LIN {X 0,Y 498.78,Z 857.029,A -85,B 0,C 180,E1 14801.152,E2 14801.152} C_VEL
LIN {X 0,Y 480.822,Z 920.353,A -85,B 0,C 180,E1 14806.511,E2 14806.511} C_VEL
LIN {X 0,Y 463.831,Z 974.464,A -85,B 0,C 180,E1 14813.724,E2 14813.724} C_VEL
LIN {X 0,Y 451.235,Z 1016.767,A -85,B 0,C 180,E1 14822.478,E2 14822.478} C_VEL
LIN {X 0,Y 444.81,Z 1044.673,A -85,B 0,C 180,E1 14831.852,E2 14831.852} C_VEL
LIN {X 0,Y 443.283,Z 1056.769,A -85,B 0,C 180,E1 14839.155,E2 14839.155} C_VEL
LIN {X 0,Y 443.188,Z 1061.056,A -85,B 0,C 180,E1 14847.74,E2 14847.74} C_VEL
LIN {X 0,Y 443.49,Z 1055.308,A -85,B 0,C 180,E1 14855.887,E2 14855.887} C_VEL
LIN {X 0,Y 445.923,Z 1037.781,A -85,B 0,C 180,E1 14864.776,E2 14864.776} C_VEL
LIN {X 0,Y 454.067,Z 1004.775,A -85,B 0,C 180,E1 14874.148,E2 14874.148} C_VEL
LIN {X 0,Y 467.703,Z 958.825,A -85,B 0,C 180,E1 14882.342,E2 14882.342} C_VEL
LIN {X 0,Y 484.897,Z 900.577,A -85,B 0,C 180,E1 14889.005,E2 14889.005} C_VEL
LIN {X 0,Y 501.352,Z 834.705,A -85,B 0,C 180,E1 14893.779,E2 14893.779} C_VEL
LIN {X 0,Y 509.754,Z 781.732,A -85,B 0,C 180,E1 14896.414,E2 14896.414} C_VEL
LIN {X 0,Y 485.015,Z 728.25,A -85,B 0,C 180,E1 14902.556,E2 14902.556} C_VEL
LIN {X 0,Y 455.384,Z 683.445,A -85,B 0,C 180,E1 14909.799,E2 14909.799} C_VEL
LIN {X 0,Y 441.694,Z 663.19,A -85,B 0,C 180,E1 14914.159,E2 14914.159} C_VEL
LIN {X 0,Y 442.478,Z 663.19,A -85,B 0,C 180,E1 14925.114,E2 14925.114} C_VEL
LIN {X 0,Y 442.609,Z 663.19,A -85,B 0,C 180,E1 14929.547,E2 14929.547} C_VEL
LIN {X 0,Y 434.436,Z 663.19,A -85,B 0,C 180,E1 14934.054,E2 14934.054} C_VEL
LIN {X 0,Y 434.643,Z 663.19,A -85,B 0,C 180,E1 14943.024,E2 14943.024} C_VEL
LIN {X 0,Y 434.152,Z 663.19,A -85,B 0,C 180,E1 14953.157,E2 14953.157} C_VEL
LIN {X 0,Y 433.829,Z 664.9,A -85,B 0,C 180,E1 14960.435,E2 14960.435} C_VEL
LIN {X 0,Y 463.212,Z 704.391,A -85,B 0,C 180,E1 14969.385,E2 14969.385} C_VEL
LIN {X 0,Y 491.827,Z 754.152,A -85,B 0,C 180,E1 14976.332,E2 14976.332} C_VEL
LIN {X 0,Y 505.339,Z 789.902,A -85,B 0,C 180,E1 14980.076,E2 14980.076} C_VEL
LIN {X 0,Y 490.914,Z 859.853,A -85,B 0,C 180,E1 14983.564,E2 14983.564} C_VEL
LIN {X 0,Y 473.096,Z 925.13,A -85,B 0,C 180,E1 14988.962,E2 14988.962} C_VEL
LIN {X 0,Y 456.226,Z 980.153,A -85,B 0,C 180,E1 14996.149,E2 14996.149} C_VEL
LIN {X 0,Y 443.812,Z 1022.566,A -85,B 0,C 180,E1 15004.717,E2 15004.717} C_VEL
LIN {X 0,Y 436.833,Z 1052.193,A -85,B 0,C 180,E1 15014.394,E2 15014.394} C_VEL
LIN {X 0,Y 435.277,Z 1066.186,A -85,B 0,C 180,E1 15022.997,E2 15022.997} C_VEL
LIN {X 0,Y 435.491,Z 1069.578,A -85,B 0,C 180,E1 15030.998,E2 15030.998} C_VEL
LIN {X 0,Y 435.549,Z 1062.657,A -85,B 0,C 180,E1 15040.026,E2 15040.026} C_VEL
LIN {X 0,Y 439.139,Z 1042.2,A -85,B 0,C 180,E1 15049.675,E2 15049.675} C_VEL
LIN {X 0,Y 448.991,Z 1006.051,A -85,B 0,C 180,E1 15059.323,E2 15059.323} C_VEL
LIN {X 0,Y 464.337,Z 958.152,A -85,B 0,C 180,E1 15067.421,E2 15067.421} C_VEL
LIN {X 0,Y 482.711,Z 899.542,A -85,B 0,C 180,E1 15073.825,E2 15073.825} C_VEL
LIN {X 0,Y 500.489,Z 832.188,A -85,B 0,C 180,E1 15078.418,E2 15078.418} C_VEL
LIN {X 0,Y 508.3,Z 786.213,A -85,B 0,C 180,E1 15080.591,E2 15080.591} C_VEL
LIN {X 0,Y 484.766,Z 736.368,A -85,B 0,C 180,E1 15087.094,E2 15087.094} C_VEL
LIN {X 0,Y 459.06,Z 697.737,A -85,B 0,C 180,E1 15094.521,E2 15094.521} C_VEL
LIN {X 0,Y 442.234,Z 676.205,A -85,B 0,C 180,E1 15101.078,E2 15101.078} C_VEL
LIN {X 0,Y 436.452,Z 669.072,A -85,B 0,C 180,E1 15104.118,E2 15104.118} C_VEL
LIN {X 0,Y 434.075,Z 663.19,A -85,B 0,C 180,E1 15106.326,E2 15106.326} C_VEL
LIN {X 0,Y 434.65,Z 663.19,A -85,B 0,C 180,E1 15116.976,E2 15116.976} C_VEL
LIN {X 0,Y 434.433,Z 663.19,A -85,B 0,C 180,E1 15125.837,E2 15125.837} C_VEL
LIN {X 0,Y 434.503,Z 665.136,A -85,B 0,C 180,E1 15131.669,E2 15131.669} C_VEL
LIN {X 0,Y 447.525,Z 682.237,A -85,B 0,C 180,E1 15138.325,E2 15138.325} C_VEL
LIN {X 0,Y 470.261,Z 712.636,A -85,B 0,C 180,E1 15146.001,E2 15146.001} C_VEL
LIN {X 0,Y 495.719,Z 757.278,A -85,B 0,C 180,E1 15153.091,E2 15153.091} C_VEL
LIN {X 0,Y 507.94,Z 791.531,A -85,B 0,C 180,E1 15157.02,E2 15157.02} C_VEL
LIN {X 0,Y 492.588,Z 859.65,A -85,B 0,C 180,E1 15160.625,E2 15160.625} C_VEL
LIN {X 0,Y 474.034,Z 922.35,A -85,B 0,C 180,E1 15166.06,E2 15166.06} C_VEL
LIN {X 0,Y 456.421,Z 976.246,A -85,B 0,C 180,E1 15173.424,E2 15173.424} C_VEL
LIN {X 0,Y 443.207,Z 1018.661,A -85,B 0,C 180,E1 15182.49,E2 15182.49} C_VEL
LIN {X 0,Y 436.635,Z 1046.422,A -85,B 0,C 180,E1 15192.309,E2 15192.309} C_VEL
LIN {X 0,Y 435.14,Z 1058.726,A -85,B 0,C 180,E1 15200.977,E2 15200.977} C_VEL
LIN {X 0,Y 435.281,Z 1060.917,A -85,B 0,C 180,E1 15209.001,E2 15209.001} C_VEL
LIN {X 0,Y 435.779,Z 1052.584,A -85,B 0,C 180,E1 15218.001,E2 15218.001} C_VEL
LIN {X 0,Y 440.317,Z 1029.675,A -85,B 0,C 180,E1 15227.941,E2 15227.941} C_VEL
LIN {X 0,Y 450.604,Z 992.208,A -85,B 0,C 180,E1 15237.291,E2 15237.291} C_VEL
LIN {X 0,Y 466.318,Z 941.94,A -85,B 0,C 180,E1 15245.186,E2 15245.186} C_VEL
LIN {X 0,Y 484.277,Z 880.392,A -85,B 0,C 180,E1 15251.389,E2 15251.389} C_VEL
LIN {X 0,Y 500.471,Z 812.301,A -85,B 0,C 180,E1 15255.622,E2 15255.622} C_VEL
LIN {X 0,Y 503.68,Z 784.382,A -85,B 0,C 180,E1 15257.043,E2 15257.043} C_VEL
LIN {X 0,Y 480.044,Z 732.332,A -85,B 0,C 180,E1 15263.229,E2 15263.229} C_VEL
LIN {X 0,Y 451.395,Z 688.691,A -85,B 0,C 180,E1 15270.571,E2 15270.571} C_VEL
LIN {X 0,Y 433.747,Z 663.19,A -85,B 0,C 180,E1 15276.72,E2 15276.72} C_VEL
LIN {X 0,Y 434.648,Z 663.19,A -85,B 0,C 180,E1 15286.903,E2 15286.903} C_VEL
LIN {X 0,Y 434.436,Z 663.19,A -85,B 0,C 180,E1 15294.054,E2 15294.054} C_VEL
LIN {X 0,Y 426.744,Z 663.19,A -85,B 0,C 180,E1 15298.697,E2 15298.697} C_VEL
LIN {X 0,Y 426.485,Z 663.19,A -85,B 0,C 180,E1 15307.178,E2 15307.178} C_VEL
LIN {X 0,Y 425.974,Z 665.123,A -85,B 0,C 180,E1 15317.653,E2 15317.653} C_VEL
LIN {X 0,Y 448.471,Z 695.077,A -85,B 0,C 180,E1 15325.749,E2 15325.749} C_VEL
LIN {X 0,Y 474.865,Z 735.267,A -85,B 0,C 180,E1 15332.732,E2 15332.732} C_VEL
LIN {X 0,Y 498.15,Z 786.178,A -85,B 0,C 180,E1 15338.91,E2 15338.91} C_VEL
LIN {X 0,Y 498.656,Z 798.243,A -85,B 0,C 180,E1 15339.698,E2 15339.698} C_VEL
LIN {X 0,Y 483.298,Z 867.659,A -85,B 0,C 180,E1 15343.412,E2 15343.412} C_VEL
LIN {X 0,Y 465.118,Z 930.433,A -85,B 0,C 180,E1 15348.904,E2 15348.904} C_VEL
LIN {X 0,Y 447.9,Z 984.105,A -85,B 0,C 180,E1 15356.257,E2 15356.257} C_VEL
LIN {X 0,Y 435.152,Z 1026.238,A -85,B 0,C 180,E1 15365.249,E2 15365.249} C_VEL
LIN {X 0,Y 428.705,Z 1053.233,A -85,B 0,C 180,E1 15374.616,E2 15374.616} C_VEL
LIN {X 0,Y 427.272,Z 1066.093,A -85,B 0,C 180,E1 15382.865,E2 15382.865} C_VEL
LIN {X 0,Y 427.503,Z 1069.503,A -85,B 0,C 180,E1 15391.017,E2 15391.017} C_VEL
LIN {X 0,Y 427.571,Z 1062.604,A -85,B 0,C 180,E1 15400.215,E2 15400.215} C_VEL
LIN {X 0,Y 431.395,Z 1042.278,A -85,B 0,C 180,E1 15410.009,E2 15410.009} C_VEL
LIN {X 0,Y 441.734,Z 1006.072,A -85,B 0,C 180,E1 15419.853,E2 15419.853} C_VEL
LIN {X 0,Y 458.167,Z 957.186,A -85,B 0,C 180,E1 15428.193,E2 15428.193} C_VEL
LIN {X 0,Y 477.4,Z 897.844,A -85,B 0,C 180,E1 15434.675,E2 15434.675} C_VEL
LIN {X 0,Y 495.435,Z 831.195,A -85,B 0,C 180,E1 15439.185,E2 15439.185} C_VEL
LIN {X 0,Y 502.744,Z 789.669,A -85,B 0,C 180,E1 15441.181,E2 15441.181} C_VEL
LIN {X 0,Y 479.872,Z 740.348,A -85,B 0,C 180,E1 15447.876,E2 15447.876} C_VEL
LIN {X 0,Y 455.268,Z 702.676,A -85,B 0,C 180,E1 15455.415,E2 15455.415} C_VEL
LIN {X 0,Y 436.885,Z 678.131,A -85,B 0,C 180,E1 15463.336,E2 15463.336} C_VEL
LIN {X 0,Y 429.602,Z 669.753,A -85,B 0,C 180,E1 15468.168,E2 15468.168} C_VEL
LIN {X 0,Y 426.492,Z 663.19,A -85,B 0,C 180,E1 15472.823,E2 15472.823} C_VEL
LIN {X 0,Y 426.967,Z 663.19,A -85,B 0,C 180,E1 15483.034,E2 15483.034} C_VEL
LIN {X 0,Y 426.767,Z 665.544,A -85,B 0,C 180,E1 15486.09,E2 15486.09} C_VEL
LIN {X 0,Y 433.558,Z 674.22,A -85,B 0,C 180,E1 15491.782,E2 15491.782} C_VEL
LIN {X 0,Y 445.568,Z 689.42,A -85,B 0,C 180,E1 15497.959,E2 15497.959} C_VEL
LIN {X 0,Y 468.291,Z 720.914,A -85,B 0,C 180,E1 15505.861,E2 15505.861} C_VEL
LIN {X 0,Y 492.084,Z 764.56,A -85,B 0,C 180,E1 15512.908,E2 15512.908} C_VEL
LIN {X 0,Y 502.331,Z 794.471,A -85,B 0,C 180,E1 15516.421,E2 15516.421} C_VEL
LIN {X 0,Y 486.135,Z 863.156,A -85,B 0,C 180,E1 15520.16,E2 15520.16} C_VEL
LIN {X 0,Y 466.596,Z 926.451,A -85,B 0,C 180,E1 15525.836,E2 15525.836} C_VEL
LIN {X 0,Y 448.604,Z 979.206,A -85,B 0,C 180,E1 15533.316,E2 15533.316} C_VEL
LIN {X 0,Y 435.185,Z 1020.487,A -85,B 0,C 180,E1 15542.49,E2 15542.49} C_VEL
LIN {X 0,Y 428.578,Z 1047.393,A -85,B 0,C 180,E1 15552.497,E2 15552.497} C_VEL
LIN {X 0,Y 427.138,Z 1058.771,A -85,B 0,C 180,E1 15560.807,E2 15560.807} C_VEL
LIN {X 0,Y 427.294,Z 1061.002,A -85,B 0,C 180,E1 15568.983,E2 15568.983} C_VEL
LIN {X 0,Y 427.826,Z 1052.724,A -85,B 0,C 180,E1 15578.15,E2 15578.15} C_VEL
LIN {X 0,Y 432.49,Z 1030.138,A -85,B 0,C 180,E1 15588.183,E2 15588.183} C_VEL
LIN {X 0,Y 442.958,Z 993.681,A -85,B 0,C 180,E1 15597.526,E2 15597.526} C_VEL
LIN {X 0,Y 458.683,Z 945.619,A -85,B 0,C 180,E1 15605.348,E2 15605.348} C_VEL
LIN {X 0,Y 476.882,Z 885.865,A -85,B 0,C 180,E1 15611.617,E2 15611.617} C_VEL
LIN {X 0,Y 494.078,Z 817.022,A -85,B 0,C 180,E1 15616.078,E2 15616.078} C_VEL
LIN {X 0,Y 497.877,Z 787.864,A -85,B 0,C 180,E1 15617.608,E2 15617.608} C_VEL
LIN {X 0,Y 475.449,Z 737.244,A -85,B 0,C 180,E1 15623.826,E2 15623.826} C_VEL
LIN {X 0,Y 446.571,Z 691.869,A -85,B 0,C 180,E1 15631.661,E2 15631.661} C_VEL
LIN {X 0,Y 428.138,Z 668.883,A -85,B 0,C 180,E1 15638.17,E2 15638.17} C_VEL
LIN {X 0,Y 425.795,Z 663.19,A -85,B 0,C 180,E1 15639.686,E2 15639.686} C_VEL
LIN {X 0,Y 426.677,Z 663.19,A -85,B 0,C 180,E1 15648.74,E2 15648.74} C_VEL
LIN {X 0,Y 426.744,Z 663.19,A -85,B 0,C 180,E1 15658.697,E2 15658.697} C_VEL
LIN {X 0,Y 418.627,Z 663.19,A -85,B 0,C 180,E1 15663.379,E2 15663.379} C_VEL
LIN {X 0,Y 418.152,Z 664.953,A -85,B 0,C 180,E1 15674.273,E2 15674.273} C_VEL
LIN {X 0,Y 436.427,Z 689.311,A -85,B 0,C 180,E1 15682.264,E2 15682.264} C_VEL
LIN {X 0,Y 462.637,Z 726.523,A -85,B 0,C 180,E1 15690.038,E2 15690.038} C_VEL
LIN {X 0,Y 487.402,Z 776.2,A -85,B 0,C 180,E1 15696.802,E2 15696.802} C_VEL
LIN {X 0,Y 493.513,Z 797.499,A -85,B 0,C 180,E1 15698.963,E2 15698.963} C_VEL
LIN {X 0,Y 477.824,Z 866.764,A -85,B 0,C 180,E1 15702.657,E2 15702.657} C_VEL
LIN {X 0,Y 458.773,Z 930.381,A -85,B 0,C 180,E1 15708.243,E2 15708.243} C_VEL
LIN {X 0,Y 440.535,Z 985.235,A -85,B 0,C 180,E1 15715.885,E2 15715.885} C_VEL
LIN {X 0,Y 427.488,Z 1026.605,A -85,B 0,C 180,E1 15724.925,E2 15724.925} C_VEL
LIN {X 0,Y 420.634,Z 1054.271,A -85,B 0,C 180,E1 15734.849,E2 15734.849} C_VEL
LIN {X 0,Y 419.279,Z 1066,A -85,B 0,C 180,E1 15742.728,E2 15742.728} C_VEL
LIN {X 0,Y 419.491,Z 1069.428,A -85,B 0,C 180,E1 15751.036,E2 15751.036} C_VEL
LIN {X 0,Y 419.619,Z 1062.554,A -85,B 0,C 180,E1 15760.41,E2 15760.41} C_VEL
LIN {X 0,Y 423.642,Z 1042.363,A -85,B 0,C 180,E1 15770.355,E2 15770.355} C_VEL
LIN {X 0,Y 434.139,Z 1007.297,A -85,B 0,C 180,E1 15780.14,E2 15780.14} C_VEL
LIN {X 0,Y 451.184,Z 958.707,A -85,B 0,C 180,E1 15788.64,E2 15788.64} C_VEL
LIN {X 0,Y 471.074,Z 899.714,A -85,B 0,C 180,E1 15795.218,E2 15795.218} C_VEL
LIN {X 0,Y 490.205,Z 831.579,A -85,B 0,C 180,E1 15799.893,E2 15799.893} C_VEL
LIN {X 0,Y 497.337,Z 793.409,A -85,B 0,C 180,E1 15801.752,E2 15801.752} C_VEL
LIN {X 0,Y 474.61,Z 743.426,A -85,B 0,C 180,E1 15808.811,E2 15808.811} C_VEL
LIN {X 0,Y 450.499,Z 706.201,A -85,B 0,C 180,E1 15816.723,E2 15816.723} C_VEL
LIN {X 0,Y 434.137,Z 684.921,A -85,B 0,C 180,E1 15824.274,E2 15824.274} C_VEL
LIN {X 0,Y 428.274,Z 677.491,A -85,B 0,C 180,E1 15828.434,E2 15828.434} C_VEL
LIN {X 0,Y 423.877,Z 670.721,A -85,B 0,C 180,E1 15833.811,E2 15833.811} C_VEL
LIN {X 0,Y 425.501,Z 672.996,A -85,B 0,C 180,E1 15845.736,E2 15845.736} C_VEL
LIN {X 0,Y 432.732,Z 682.917,A -85,B 0,C 180,E1 15851.934,E2 15851.934} C_VEL
LIN {X 0,Y 447.738,Z 701.689,A -85,B 0,C 180,E1 15859.278,E2 15859.278} C_VEL
LIN {X 0,Y 471.802,Z 738.399,A -85,B 0,C 180,E1 15867.522,E2 15867.522} C_VEL
LIN {X 0,Y 493.23,Z 784.173,A -85,B 0,C 180,E1 15874.336,E2 15874.336} C_VEL
LIN {X 0,Y 496.572,Z 798.512,A -85,B 0,C 180,E1 15875.861,E2 15875.861} C_VEL
LIN {X 0,Y 479.996,Z 865.734,A -85,B 0,C 180,E1 15879.618,E2 15879.618} C_VEL
LIN {X 0,Y 459.786,Z 928.731,A -85,B 0,C 180,E1 15885.396,E2 15885.396} C_VEL
LIN {X 0,Y 441.159,Z 981.112,A -85,B 0,C 180,E1 15893.02,E2 15893.02} C_VEL
LIN {X 0,Y 427.338,Z 1021.674,A -85,B 0,C 180,E1 15902.347,E2 15902.347} C_VEL
LIN {X 0,Y 420.72,Z 1047.399,A -85,B 0,C 180,E1 15912.159,E2 15912.159} C_VEL
LIN {X 0,Y 419.138,Z 1058.816,A -85,B 0,C 180,E1 15920.63,E2 15920.63} C_VEL
LIN {X 0,Y 419.29,Z 1061.086,A -85,B 0,C 180,E1 15928.963,E2 15928.963} C_VEL
LIN {X 0,Y 419.893,Z 1052.861,A -85,B 0,C 180,E1 15938.305,E2 15938.305} C_VEL
LIN {X 0,Y 424.578,Z 1031.01,A -85,B 0,C 180,E1 15948.292,E2 15948.292} C_VEL
LIN {X 0,Y 435.694,Z 993.933,A -85,B 0,C 180,E1 15958.025,E2 15958.025} C_VEL
LIN {X 0,Y 452.484,Z 944.571,A -85,B 0,C 180,E1 15966.125,E2 15966.125} C_VEL
LIN {X 0,Y 471.328,Z 884.634,A -85,B 0,C 180,E1 15972.411,E2 15972.411} C_VEL
LIN {X 0,Y 488.788,Z 816.604,A -85,B 0,C 180,E1 15976.807,E2 15976.807} C_VEL
LIN {X 0,Y 492.112,Z 791.275,A -85,B 0,C 180,E1 15978.192,E2 15978.192} C_VEL
LIN {X 0,Y 470.456,Z 741.37,A -85,B 0,C 180,E1 15984.524,E2 15984.524} C_VEL
LIN {X 0,Y 443.694,Z 698.608,A -85,B 0,C 180,E1 15992.168,E2 15992.168} C_VEL
LIN {X 0,Y 422.122,Z 670.229,A -85,B 0,C 180,E1 16000.454,E2 16000.454} C_VEL
LIN {X 0,Y 418.095,Z 663.19,A -85,B 0,C 180,E1 16003.048,E2 16003.048} C_VEL
LIN {X 0,Y 418.386,Z 663.19,A -85,B 0,C 180,E1 16012.728,E2 16012.728} C_VEL
LIN {X 0,Y 418.464,Z 663.19,A -85,B 0,C 180,E1 16021.062,E2 16021.062} C_VEL
LIN {X 0,Y 418.627,Z 663.19,A -85,B 0,C 180,E1 16023.379,E2 16023.379} C_VEL
LIN {X 0,Y 410.326,Z 663.19,A -85,B 0,C 180,E1 16028.157,E2 16028.157} C_VEL
LIN {X 0,Y 410.695,Z 666.004,A -85,B 0,C 180,E1 16030.134,E2 16030.134} C_VEL
LIN {X 0,Y 417.572,Z 674.992,A -85,B 0,C 180,E1 16034.609,E2 16034.609} C_VEL
LIN {X 0,Y 433.792,Z 695.796,A -85,B 0,C 180,E1 16041.729,E2 16041.729} C_VEL
LIN {X 0,Y 459.528,Z 733.457,A -85,B 0,C 180,E1 16049.722,E2 16049.722} C_VEL
LIN {X 0,Y 482.731,Z 781.872,A -85,B 0,C 180,E1 16056.428,E2 16056.428} C_VEL
LIN {X 0,Y 487.905,Z 799.598,A -85,B 0,C 180,E1 16058.33,E2 16058.33} C_VEL
LIN {X 0,Y 471.492,Z 869.149,A -85,B 0,C 180,E1 16062.121,E2 16062.121} C_VEL
LIN {X 0,Y 451.706,Z 932.866,A -85,B 0,C 180,E1 16067.86,E2 16067.86} C_VEL
LIN {X 0,Y 432.989,Z 986.936,A -85,B 0,C 180,E1 16075.601,E2 16075.601} C_VEL
LIN {X 0,Y 419.444,Z 1028.165,A -85,B 0,C 180,E1 16084.923,E2 16084.923} C_VEL
LIN {X 0,Y 412.534,Z 1055.151,A -85,B 0,C 180,E1 16095.09,E2 16095.09} C_VEL
LIN {X 0,Y 411.199,Z 1067.647,A -85,B 0,C 180,E1 16104.711,E2 16104.711} C_VEL
LIN {X 0,Y 411.152,Z 1068.842,A -85,B 0,C 180,E1 16113.172,E2 16113.172} C_VEL
LIN {X 0,Y 412.384,Z 1058.853,A -85,B 0,C 180,E1 16123.08,E2 16123.08} C_VEL
LIN {X 0,Y 417.766,Z 1034.302,A -85,B 0,C 180,E1 16133.534,E2 16133.534} C_VEL
LIN {X 0,Y 430.738,Z 996.165,A -85,B 0,C 180,E1 16143.071,E2 16143.071} C_VEL
LIN {X 0,Y 450.189,Z 943.725,A -85,B 0,C 180,E1 16151.313,E2 16151.313} C_VEL
LIN {X 0,Y 470.83,Z 882.841,A -85,B 0,C 180,E1 16157.342,E2 16157.342} C_VEL
LIN {X 0,Y 489.351,Z 812.57,A -85,B 0,C 180,E1 16161.584,E2 16161.584} C_VEL
LIN {X 0,Y 491.697,Z 796.347,A -85,B 0,C 180,E1 16162.434,E2 16162.434} C_VEL
LIN {X 0,Y 469.974,Z 748.012,A -85,B 0,C 180,E1 16169.534,E2 16169.534} C_VEL
LIN {X 0,Y 447.711,Z 712.682,A -85,B 0,C 180,E1 16177.295,E2 16177.295} C_VEL
LIN {X 0,Y 431.971,Z 691.832,A -85,B 0,C 180,E1 16184.959,E2 16184.959} C_VEL
LIN {X 0,Y 426.531,Z 684.771,A -85,B 0,C 180,E1 16189.081,E2 16189.081} C_VEL
LIN {X 0,Y 422.626,Z 678.518,A -85,B 0,C 180,E1 16194.31,E2 16194.31} C_VEL
LIN {X 0,Y 424.354,Z 680.93,A -85,B 0,C 180,E1 16205.558,E2 16205.558} C_VEL
LIN {X 0,Y 432.326,Z 691.884,A -85,B 0,C 180,E1 16212.331,E2 16212.331} C_VEL
LIN {X 0,Y 447.389,Z 711.911,A -85,B 0,C 180,E1 16219.68,E2 16219.68} C_VEL
LIN {X 0,Y 469.419,Z 746.964,A -85,B 0,C 180,E1 16227.508,E2 16227.508} C_VEL
LIN {X 0,Y 489.261,Z 791.653,A -85,B 0,C 180,E1 16234.198,E2 16234.198} C_VEL
LIN {X 0,Y 490.644,Z 803.508,A -85,B 0,C 180,E1 16235.326,E2 16235.326} C_VEL
LIN {X 0,Y 473.328,Z 870.264,A -85,B 0,C 180,E1 16239.203,E2 16239.203} C_VEL
LIN {X 0,Y 452.36,Z 932.822,A -85,B 0,C 180,E1 16245.151,E2 16245.151} C_VEL
LIN {X 0,Y 433.01,Z 984.809,A -85,B 0,C 180,E1 16253.078,E2 16253.078} C_VEL
LIN {X 0,Y 419.173,Z 1023.727,A -85,B 0,C 180,E1 16262.465,E2 16262.465} C_VEL
LIN {X 0,Y 412.585,Z 1048.87,A -85,B 0,C 180,E1 16272.634,E2 16272.634} C_VEL
LIN {X 0,Y 411.141,Z 1058.862,A -85,B 0,C 180,E1 16280.446,E2 16280.446} C_VEL
LIN {X 0,Y 411.285,Z 1061.171,A -85,B 0,C 180,E1 16288.943,E2 16288.943} C_VEL
LIN {X 0,Y 411.961,Z 1052.997,A -85,B 0,C 180,E1 16298.466,E2 16298.466} C_VEL
LIN {X 0,Y 416.812,Z 1031.202,A -85,B 0,C 180,E1 16308.645,E2 16308.645} C_VEL
LIN {X 0,Y 428.484,Z 994.183,A -85,B 0,C 180,E1 16318.539,E2 16318.539} C_VEL
LIN {X 0,Y 445.848,Z 945.171,A -85,B 0,C 180,E1 16326.709,E2 16326.709} C_VEL
LIN {X 0,Y 465.527,Z 884.677,A -85,B 0,C 180,E1 16333.114,E2 16333.114} C_VEL
LIN {X 0,Y 483.714,Z 815.532,A -85,B 0,C 180,E1 16337.586,E2 16337.586} C_VEL
LIN {X 0,Y 486.452,Z 795.07,A -85,B 0,C 180,E1 16338.728,E2 16338.728} C_VEL
LIN {X 0,Y 465.506,Z 745.361,A -85,B 0,C 180,E1 16345.233,E2 16345.233} C_VEL
LIN {X 0,Y 440.008,Z 704.189,A -85,B 0,C 180,E1 16352.948,E2 16352.948} C_VEL
LIN {X 0,Y 420.1,Z 677.619,A -85,B 0,C 180,E1 16360.911,E2 16360.911} C_VEL
LIN {X 0,Y 413.018,Z 669.205,A -85,B 0,C 180,E1 16364.981,E2 16364.981} C_VEL
LIN {X 0,Y 410.543,Z 663.19,A -85,B 0,C 180,E1 16367.316,E2 16367.316} C_VEL
LIN {X 0,Y 410.76,Z 663.19,A -85,B 0,C 180,E1 16378.964,E2 16378.964} C_VEL
LIN {X 0,Y 410.326,Z 663.19,A -85,B 0,C 180,E1 16388.157,E2 16388.157} C_VEL
LIN {X 0,Y 410.731,Z 676.091,A -85,B 0,C 180,E1 16390.981,E2 16390.981} C_VEL
LIN {X 0,Y 420.44,Z 687.719,A -85,B 0,C 180,E1 16396.607,E2 16396.607} C_VEL
LIN {X 0,Y 443.836,Z 719.972,A -85,B 0,C 180,E1 16405.533,E2 16405.533} C_VEL
LIN {X 0,Y 467.876,Z 762.883,A -85,B 0,C 180,E1 16412.837,E2 16412.837} C_VEL
LIN {X 0,Y 482.174,Z 802.573,A -85,B 0,C 180,E1 16417.725,E2 16417.725} C_VEL
LIN {X 0,Y 465.103,Z 871.898,A -85,B 0,C 180,E1 16421.598,E2 16421.598} C_VEL
LIN {X 0,Y 444.653,Z 935.254,A -85,B 0,C 180,E1 16427.449,E2 16427.449} C_VEL
LIN {X 0,Y 425.464,Z 988.588,A -85,B 0,C 180,E1 16435.297,E2 16435.297} C_VEL
LIN {X 0,Y 411.411,Z 1029.584,A -85,B 0,C 180,E1 16444.921,E2 16444.921} C_VEL
LIN {X 0,Y 404.653,Z 1055.033,A -85,B 0,C 180,E1 16454.793,E2 16454.793} C_VEL
LIN {X 0,Y 403.207,Z 1067.552,A -85,B 0,C 180,E1 16464.605,E2 16464.605} C_VEL
LIN {X 0,Y 403.122,Z 1068.654,A -85,B 0,C 180,E1 16473.483,E2 16473.483} C_VEL
LIN {X 0,Y 404.467,Z 1058.614,A -85,B 0,C 180,E1 16483.455,E2 16483.455} C_VEL
LIN {X 0,Y 410.185,Z 1034.297,A -85,B 0,C 180,E1 16493.996,E2 16493.996} C_VEL
LIN {X 0,Y 423.8,Z 996.205,A -85,B 0,C 180,E1 16503.684,E2 16503.684} C_VEL
LIN {X 0,Y 443.931,Z 944.043,A -85,B 0,C 180,E1 16511.989,E2 16511.989} C_VEL
LIN {X 0,Y 465.564,Z 882.508,A -85,B 0,C 180,E1 16518.116,E2 16518.116} C_VEL
LIN {X 0,Y 484.304,Z 813.467,A -85,B 0,C 180,E1 16522.305,E2 16522.305} C_VEL
LIN {X 0,Y 486.328,Z 800.34,A -85,B 0,C 180,E1 16522.999,E2 16522.999} C_VEL
LIN {X 0,Y 465.605,Z 752.891,A -85,B 0,C 180,E1 16530.207,E2 16530.207} C_VEL
LIN {X 0,Y 444.55,Z 718.47,A -85,B 0,C 180,E1 16538.05,E2 16538.05} C_VEL
LIN {X 0,Y 427.604,Z 694.207,A -85,B 0,C 180,E1 16547.425,E2 16547.425} C_VEL
LIN {X 0,Y 421.409,Z 686.303,A -85,B 0,C 180,E1 16554.812,E2 16554.812} C_VEL
LIN {X 0,Y 423.218,Z 688.807,A -85,B 0,C 180,E1 16565.379,E2 16565.379} C_VEL
LIN {X 0,Y 433.701,Z 702.296,A -85,B 0,C 180,E1 16573.706,E2 16573.706} C_VEL
LIN {X 0,Y 453.095,Z 731.195,A -85,B 0,C 180,E1 16582.505,E2 16582.505} C_VEL
LIN {X 0,Y 474.432,Z 771.075,A -85,B 0,C 180,E1 16590.101,E2 16590.101} C_VEL
LIN {X 0,Y 485.587,Z 804.638,A -85,B 0,C 180,E1 16594.61,E2 16594.61} C_VEL
LIN {X 0,Y 467.66,Z 871.488,A -85,B 0,C 180,E1 16598.531,E2 16598.531} C_VEL
LIN {X 0,Y 446.2,Z 933.313,A -85,B 0,C 180,E1 16604.475,E2 16604.475} C_VEL
LIN {X 0,Y 426.147,Z 985.009,A -85,B 0,C 180,E1 16612.456,E2 16612.456} C_VEL
LIN {X 0,Y 411.786,Z 1023.681,A -85,B 0,C 180,E1 16621.928,E2 16621.928} C_VEL
LIN {X 0,Y 404.717,Z 1048.925,A -85,B 0,C 180,E1 16632.312,E2 16632.312} C_VEL
LIN {X 0,Y 402.974,Z 1060.342,A -85,B 0,C 180,E1 16642.431,E2 16642.431} C_VEL
LIN {X 0,Y 403.105,Z 1060.411,A -85,B 0,C 180,E1 16651.077,E2 16651.077} C_VEL
LIN {X 0,Y 404.769,Z 1049.772,A -85,B 0,C 180,E1 16660.796,E2 16660.796} C_VEL
LIN {X 0,Y 410.596,Z 1025.231,A -85,B 0,C 180,E1 16671.105,E2 16671.105} C_VEL
LIN {X 0,Y 423.742,Z 987.027,A -85,B 0,C 180,E1 16680.596,E2 16680.596} C_VEL
LIN {X 0,Y 442.82,Z 935.693,A -85,B 0,C 180,E1 16688.611,E2 16688.611} C_VEL
LIN {X 0,Y 462.857,Z 875.092,A -85,B 0,C 180,E1 16694.614,E2 16694.614} C_VEL
LIN {X 0,Y 480.805,Z 804.571,A -85,B 0,C 180,E1 16698.855,E2 16698.855} C_VEL
LIN {X 0,Y 473.443,Z 777.578,A -85,B 0,C 180,E1 16701.918,E2 16701.918} C_VEL
LIN {X 0,Y 449.835,Z 730.158,A -85,B 0,C 180,E1 16709.29,E2 16709.29} C_VEL
LIN {X 0,Y 425.035,Z 693.221,A -85,B 0,C 180,E1 16718.14,E2 16718.14} C_VEL
LIN {X 0,Y 411.665,Z 676.93,A -85,B 0,C 180,E1 16725.204,E2 16725.204} C_VEL
LIN {X 0,Y 407.068,Z 670.401,A -85,B 0,C 180,E1 16729.009,E2 16729.009} C_VEL
LIN {X 0,Y 402.76,Z 663.19,A -85,B 0,C 180,E1 16738.944,E2 16738.944} C_VEL
LIN {X 0,Y 409.313,Z 673.724,A -85,B 0,C 180,E1 16749.85,E2 16749.85} C_VEL
LIN {X 0,Y 410.731,Z 676.091,A -85,B 0,C 180,E1 16750.981,E2 16750.981} C_VEL
LIN {X 0,Y 413.955,Z 689.296,A -85,B 0,C 180,E1 16753.73,E2 16753.73} C_VEL
LIN {X 0,Y 432.831,Z 714.723,A -85,B 0,C 180,E1 16762.27,E2 16762.27} C_VEL
LIN {X 0,Y 456.296,Z 753.371,A -85,B 0,C 180,E1 16770.092,E2 16770.092} C_VEL
LIN {X 0,Y 476.397,Z 803.084,A -85,B 0,C 180,E1 16776.904,E2 16776.904} C_VEL
LIN {X 0,Y 458.764,Z 874.617,A -85,B 0,C 180,E1 16781.058,E2 16781.058} C_VEL
LIN {X 0,Y 437.817,Z 937.111,A -85,B 0,C 180,E1 16786.964,E2 16786.964} C_VEL
LIN {X 0,Y 418.137,Z 989.697,A -85,B 0,C 180,E1 16794.898,E2 16794.898} C_VEL
LIN {X 0,Y 403.944,Z 1029.428,A -85,B 0,C 180,E1 16804.424,E2 16804.424} C_VEL
LIN {X 0,Y 396.793,Z 1054.914,A -85,B 0,C 180,E1 16814.484,E2 16814.484} C_VEL
LIN {X 0,Y 395.198,Z 1067.457,A -85,B 0,C 180,E1 16824.496,E2 16824.496} C_VEL
LIN {X 0,Y 395.164,Z 1068.706,A -85,B 0,C 180,E1 16833.3,E2 16833.3} C_VEL
LIN {X 0,Y 396.434,Z 1059.26,A -85,B 0,C 180,E1 16843.269,E2 16843.269} C_VEL
LIN {X 0,Y 402.114,Z 1035.962,A -85,B 0,C 180,E1 16853.916,E2 16853.916} C_VEL
LIN {X 0,Y 416.406,Z 997.571,A -85,B 0,C 180,E1 16864.05,E2 16864.05} C_VEL
LIN {X 0,Y 436.712,Z 947.032,A -85,B 0,C 180,E1 16872.338,E2 16872.338} C_VEL
LIN {X 0,Y 458.953,Z 886.124,A -85,B 0,C 180,E1 16878.6,E2 16878.6} C_VEL
LIN {X 0,Y 478.498,Z 817.793,A -85,B 0,C 180,E1 16882.876,E2 16882.876} C_VEL
LIN {X 0,Y 480.604,Z 803.229,A -85,B 0,C 180,E1 16883.719,E2 16883.719} C_VEL
LIN {X 0,Y 460.9,Z 756.777,A -85,B 0,C 180,E1 16891.051,E2 16891.051} C_VEL
LIN {X 0,Y 439.898,Z 721.858,A -85,B 0,C 180,E1 16899.53,E2 16899.53} C_VEL
LIN {X 0,Y 425.574,Z 701.589,A -85,B 0,C 180,E1 16908.207,E2 16908.207} C_VEL
LIN {X 0,Y 420.437,Z 694.25,A -85,B 0,C 180,E1 16914.799,E2 16914.799} C_VEL
LIN {X 0,Y 422.132,Z 696.769,A -85,B 0,C 180,E1 16925.264,E2 16925.264} C_VEL
LIN {X 0,Y 432.221,Z 710.344,A -85,B 0,C 180,E1 16933.56,E2 16933.56} C_VEL
LIN {X 0,Y 450.62,Z 738.529,A -85,B 0,C 180,E1 16942.239,E2 16942.239} C_VEL
LIN {X 0,Y 470.322,Z 777.205,A -85,B 0,C 180,E1 16949.724,E2 16949.724} C_VEL
LIN {X 0,Y 480.13,Z 808.043,A -85,B 0,C 180,E1 16953.982,E2 16953.982} C_VEL
LIN {X 0,Y 461.448,Z 874.696,A -85,B 0,C 180,E1 16957.989,E2 16957.989} C_VEL
LIN {X 0,Y 439.224,Z 935.955,A -85,B 0,C 180,E1 16964.059,E2 16964.059} C_VEL
LIN {X 0,Y 418.391,Z 987.576,A -85,B 0,C 180,E1 16972.293,E2 16972.293} C_VEL
LIN {X 0,Y 403.606,Z 1025.751,A -85,B 0,C 180,E1 16982.046,E2 16982.046} C_VEL
LIN {X 0,Y 396.627,Z 1050.144,A -85,B 0,C 180,E1 16992.66,E2 16992.66} C_VEL
LIN {X 0,Y 394.971,Z 1060.402,A -85,B 0,C 180,E1 17002.277,E2 17002.277} C_VEL
LIN {X 0,Y 395.123,Z 1060.507,A -85,B 0,C 180,E1 17011.099,E2 17011.099} C_VEL
LIN {X 0,Y 396.818,Z 1049.92,A -85,B 0,C 180,E1 17021.015,E2 17021.015} C_VEL
LIN {X 0,Y 402.98,Z 1025.433,A -85,B 0,C 180,E1 17031.524,E2 17031.524} C_VEL
LIN {X 0,Y 417.052,Z 986.302,A -85,B 0,C 180,E1 17041.372,E2 17041.372} C_VEL
LIN {X 0,Y 436.639,Z 935.624,A -85,B 0,C 180,E1 17049.33,E2 17049.33} C_VEL
LIN {X 0,Y 457.62,Z 874.08,A -85,B 0,C 180,E1 17055.433,E2 17055.433} C_VEL
LIN {X 0,Y 475.423,Z 803.146,A -85,B 0,C 180,E1 17059.765,E2 17059.765} C_VEL
LIN {X 0,Y 456.44,Z 755.227,A -85,B 0,C 180,E1 17066.464,E2 17066.464} C_VEL
LIN {X 0,Y 433.063,Z 715.031,A -85,B 0,C 180,E1 17074.44,E2 17074.44} C_VEL
LIN {X 0,Y 412.369,Z 686.154,A -85,B 0,C 180,E1 17084.136,E2 17084.136} C_VEL
LIN {X 0,Y 405.271,Z 677.94,A -85,B 0,C 180,E1 17089.777,E2 17089.777} C_VEL
LIN {X 0,Y 401.557,Z 671.088,A -85,B 0,C 180,E1 17098.941,E2 17098.941} C_VEL
LIN {X 0,Y 408.136,Z 681.783,A -85,B 0,C 180,E1 17109.733,E2 17109.733} C_VEL
LIN {X 0,Y 413.955,Z 689.296,A -85,B 0,C 180,E1 17113.73,E2 17113.73} C_VEL
LIN {X 0,Y 417.622,Z 703.934,A -85,B 0,C 180,E1 17116.302,E2 17116.302} C_VEL
LIN {X 0,Y 438.689,Z 734.782,A -85,B 0,C 180,E1 17124.963,E2 17124.963} C_VEL
LIN {X 0,Y 459.758,Z 775.667,A -85,B 0,C 180,E1 17132.164,E2 17132.164} C_VEL
LIN {X 0,Y 470.533,Z 810.03,A -85,B 0,C 180,E1 17136.533,E2 17136.533} C_VEL
LIN {X 0,Y 452.455,Z 877.351,A -85,B 0,C 180,E1 17140.504,E2 17140.504} C_VEL
LIN {X 0,Y 430.526,Z 940.237,A -85,B 0,C 180,E1 17146.621,E2 17146.621} C_VEL
LIN {X 0,Y 410.211,Z 992.147,A -85,B 0,C 180,E1 17154.76,E2 17154.76} C_VEL
LIN {X 0,Y 395.501,Z 1031.923,A -85,B 0,C 180,E1 17164.757,E2 17164.757} C_VEL
LIN {X 0,Y 388.473,Z 1056.745,A -85,B 0,C 180,E1 17175.302,E2 17175.302} C_VEL
LIN {X 0,Y 387.2,Z 1067.362,A -85,B 0,C 180,E1 17184.382,E2 17184.382} C_VEL
LIN {X 0,Y 387.17,Z 1068.638,A -85,B 0,C 180,E1 17193.369,E2 17193.369} C_VEL
LIN {X 0,Y 388.492,Z 1059.213,A -85,B 0,C 180,E1 17203.545,E2 17203.545} C_VEL
LIN {X 0,Y 394.819,Z 1035.088,A -85,B 0,C 180,E1 17214.714,E2 17214.714} C_VEL
LIN {X 0,Y 409.515,Z 997.615,A -85,B 0,C 180,E1 17224.704,E2 17224.704} C_VEL
LIN {X 0,Y 430.727,Z 946.955,A -85,B 0,C 180,E1 17233.1,E2 17233.1} C_VEL
LIN {X 0,Y 453.64,Z 886.311,A -85,B 0,C 180,E1 17239.367,E2 17239.367} C_VEL
LIN {X 0,Y 473.787,Z 817.738,A -85,B 0,C 180,E1 17243.671,E2 17243.671} C_VEL
LIN {X 0,Y 475.244,Z 807.109,A -85,B 0,C 180,E1 17244.324,E2 17244.324} C_VEL
LIN {X 0,Y 456.414,Z 761.304,A -85,B 0,C 180,E1 17251.839,E2 17251.839} C_VEL
LIN {X 0,Y 437.247,Z 728.652,A -85,B 0,C 180,E1 17260.063,E2 17260.063} C_VEL
LIN {X 0,Y 424.291,Z 709.408,A -85,B 0,C 180,E1 17268.369,E2 17268.369} C_VEL
LIN {X 0,Y 419.465,Z 702.198,A -85,B 0,C 180,E1 17274.787,E2 17274.787} C_VEL
LIN {X 0,Y 421.044,Z 704.712,A -85,B 0,C 180,E1 17285.148,E2 17285.148} C_VEL
LIN {X 0,Y 430.623,Z 718.146,A -85,B 0,C 180,E1 17293.351,E2 17293.351} C_VEL
LIN {X 0,Y 448.03,Z 746.062,A -85,B 0,C 180,E1 17302.045,E2 17302.045} C_VEL
LIN {X 0,Y 466.85,Z 785.129,A -85,B 0,C 180,E1 17309.654,E2 17309.654} C_VEL
LIN {X 0,Y 474.533,Z 811.829,A -85,B 0,C 180,E1 17313.361,E2 17313.361} C_VEL
LIN {X 0,Y 455.067,Z 878.138,A -85,B 0,C 180,E1 17317.466,E2 17317.466} C_VEL
LIN {X 0,Y 432.17,Z 938.734,A -85,B 0,C 180,E1 17323.642,E2 17323.642} C_VEL
LIN {X 0,Y 410.62,Z 990.147,A -85,B 0,C 180,E1 17332.123,E2 17332.123} C_VEL
LIN {X 0,Y 395.584,Z 1027.447,A -85,B 0,C 180,E1 17342.048,E2 17342.048} C_VEL
LIN {X 0,Y 388.571,Z 1051.29,A -85,B 0,C 180,E1 17352.98,E2 17352.98} C_VEL
LIN {X 0,Y 386.968,Z 1060.462,A -85,B 0,C 180,E1 17362.116,E2 17362.116} C_VEL
LIN {X 0,Y 387.146,Z 1060.603,A -85,B 0,C 180,E1 17371.122,E2 17371.122} C_VEL
LIN {X 0,Y 388.874,Z 1050.067,A -85,B 0,C 180,E1 17381.243,E2 17381.243} C_VEL
LIN {X 0,Y 395.356,Z 1025.656,A -85,B 0,C 180,E1 17391.953,E2 17391.953} C_VEL
LIN {X 0,Y 410.107,Z 986.56,A -85,B 0,C 180,E1 17401.966,E2 17401.966} C_VEL
LIN {X 0,Y 430.398,Z 935.953,A -85,B 0,C 180,E1 17410.015,E2 17410.015} C_VEL
LIN {X 0,Y 452.022,Z 874.555,A -85,B 0,C 180,E1 17416.159,E2 17416.159} C_VEL
LIN {X 0,Y 469.763,Z 806.657,A -85,B 0,C 180,E1 17420.375,E2 17420.375} C_VEL
LIN {X 0,Y 451.432,Z 758.915,A -85,B 0,C 180,E1 17427.266,E2 17427.266} C_VEL
LIN {X 0,Y 429.05,Z 719.882,A -85,B 0,C 180,E1 17435.438,E2 17435.438} C_VEL
LIN {X 0,Y 410.358,Z 693.494,A -85,B 0,C 180,E1 17444.744,E2 17444.744} C_VEL
LIN {X 0,Y 403.798,Z 685.571,A -85,B 0,C 180,E1 17450.286,E2 17450.286} C_VEL
LIN {X 0,Y 400.609,Z 679.158,A -85,B 0,C 180,E1 17459.413,E2 17459.413} C_VEL
LIN {X 0,Y 407.044,Z 689.939,A -85,B 0,C 180,E1 17469.683,E2 17469.683} C_VEL
LIN {X 0,Y 417.622,Z 703.934,A -85,B 0,C 180,E1 17476.302,E2 17476.302} C_VEL
LIN {X 0,Y 424.756,Z 724.123,A -85,B 0,C 180,E1 17480.169,E2 17480.169} C_VEL
LIN {X 0,Y 446.584,Z 761.339,A -85,B 0,C 180,E1 17488.499,E2 17488.499} C_VEL
LIN {X 0,Y 464.824,Z 808.996,A -85,B 0,C 180,E1 17495.543,E2 17495.543} C_VEL
LIN {X 0,Y 446.173,Z 880.206,A -85,B 0,C 180,E1 17499.946,E2 17499.946} C_VEL
LIN {X 0,Y 423.74,Z 941.914,A -85,B 0,C 180,E1 17506.104,E2 17506.104} C_VEL
LIN {X 0,Y 402.939,Z 993.113,A -85,B 0,C 180,E1 17514.316,E2 17514.316} C_VEL
LIN {X 0,Y 387.881,Z 1032.158,A -85,B 0,C 180,E1 17524.364,E2 17524.364} C_VEL
LIN {X 0,Y 380.578,Z 1056.624,A -85,B 0,C 180,E1 17534.99,E2 17534.99} C_VEL
LIN {X 0,Y 379.192,Z 1067.266,A -85,B 0,C 180,E1 17544.263,E2 17544.263} C_VEL
LIN {X 0,Y 379.162,Z 1068.571,A -85,B 0,C 180,E1 17553.44,E2 17553.44} C_VEL
LIN {X 0,Y 380.547,Z 1059.167,A -85,B 0,C 180,E1 17563.833,E2 17563.833} C_VEL
LIN {X 0,Y 387.222,Z 1035.318,A -85,B 0,C 180,E1 17575.145,E2 17575.145} C_VEL
LIN {X 0,Y 402.688,Z 997.661,A -85,B 0,C 180,E1 17585.379,E2 17585.379} C_VEL
LIN {X 0,Y 424.893,Z 946.703,A -85,B 0,C 180,E1 17593.907,E2 17593.907} C_VEL
LIN {X 0,Y 448.8,Z 885.452,A -85,B 0,C 180,E1 17600.236,E2 17600.236} C_VEL
LIN {X 0,Y 469.509,Z 816.341,A -85,B 0,C 180,E1 17604.55,E2 17604.55} C_VEL
LIN {X 0,Y 467.707,Z 804.309,A -85,B 0,C 180,E1 17605.933,E2 17605.933} C_VEL
LIN {X 0,Y 449.631,Z 761.277,A -85,B 0,C 180,E1 17613.597,E2 17613.597} C_VEL
LIN {X 0,Y 431.737,Z 730.643,A -85,B 0,C 180,E1 17622.194,E2 17622.194} C_VEL
LIN {X 0,Y 421.484,Z 715.897,A -85,B 0,C 180,E1 17629.867,E2 17629.867} C_VEL
LIN {X 0,Y 418.189,Z 710.027,A -85,B 0,C 180,E1 17635.227,E2 17635.227} C_VEL
LIN {X 0,Y 419.758,Z 712.603,A -85,B 0,C 180,E1 17644.998,E2 17644.998} C_VEL
LIN {X 0,Y 428.948,Z 726.059,A -85,B 0,C 180,E1 17653.209,E2 17653.209} C_VEL
LIN {X 0,Y 445.716,Z 754.015,A -85,B 0,C 180,E1 17661.976,E2 17661.976} C_VEL
LIN {X 0,Y 463.688,Z 794.108,A -85,B 0,C 180,E1 17669.753,E2 17669.753} C_VEL
LIN {X 0,Y 468.929,Z 815.8,A -85,B 0,C 180,E1 17672.748,E2 17672.748} C_VEL
LIN {X 0,Y 448.673,Z 881.759,A -85,B 0,C 180,E1 17676.95,E2 17676.95} C_VEL
LIN {X 0,Y 424.901,Z 942.169,A -85,B 0,C 180,E1 17683.304,E2 17683.304} C_VEL
LIN {X 0,Y 403.432,Z 991.383,A -85,B 0,C 180,E1 17691.669,E2 17691.669} C_VEL
LIN {X 0,Y 387.61,Z 1028.892,A -85,B 0,C 180,E1 17701.983,E2 17701.983} C_VEL
LIN {X 0,Y 380.682,Z 1051.304,A -85,B 0,C 180,E1 17712.617,E2 17712.617} C_VEL
LIN {X 0,Y 378.966,Z 1060.522,A -85,B 0,C 180,E1 17721.949,E2 17721.949} C_VEL
LIN {X 0,Y 379.17,Z 1060.698,A -85,B 0,C 180,E1 17731.145,E2 17731.145} C_VEL
LIN {X 0,Y 380.938,Z 1050.213,A -85,B 0,C 180,E1 17741.48,E2 17741.48} C_VEL
LIN {X 0,Y 387.66,Z 1026.225,A -85,B 0,C 180,E1 17752.281,E2 17752.281} C_VEL
LIN {X 0,Y 402.622,Z 988.196,A -85,B 0,C 180,E1 17762.296,E2 17762.296} C_VEL
LIN {X 0,Y 424.188,Z 936.287,A -85,B 0,C 180,E1 17770.723,E2 17770.723} C_VEL
LIN {X 0,Y 446.476,Z 875.022,A -85,B 0,C 180,E1 17776.905,E2 17776.905} C_VEL
LIN {X 0,Y 463.93,Z 809.396,A -85,B 0,C 180,E1 17781.097,E2 17781.097} C_VEL
LIN {X 0,Y 446.548,Z 763.243,A -85,B 0,C 180,E1 17788.01,E2 17788.01} C_VEL
LIN {X 0,Y 425.8,Z 725.974,A -85,B 0,C 180,E1 17796.104,E2 17796.104} C_VEL
LIN {X 0,Y 408.598,Z 700.925,A -85,B 0,C 180,E1 17805.228,E2 17805.228} C_VEL
LIN {X 0,Y 402.592,Z 693.356,A -85,B 0,C 180,E1 17810.53,E2 17810.53} C_VEL
LIN {X 0,Y 399.609,Z 687.299,A -85,B 0,C 180,E1 17819.412,E2 17819.412} C_VEL
LIN {X 0,Y 405.893,Z 697.931,A -85,B 0,C 180,E1 17829.575,E2 17829.575} C_VEL
LIN {X 0,Y 419.484,Z 716.07,A -85,B 0,C 180,E1 17837.799,E2 17837.799} C_VEL
LIN {X 0,Y 424.756,Z 724.123,A -85,B 0,C 180,E1 17840.169,E2 17840.169} C_VEL
LIN {X 0,Y 428.327,Z 740.919,A -85,B 0,C 180,E1 17842.421,E2 17842.421} C_VEL
LIN {X 0,Y 447.796,Z 779.271,A -85,B 0,C 180,E1 17850.05,E2 17850.05} C_VEL
LIN {X 0,Y 459.343,Z 816.333,A -85,B 0,C 180,E1 17855.244,E2 17855.244} C_VEL
LIN {X 0,Y 439.462,Z 884.04,A -85,B 0,C 180,E1 17859.464,E2 17859.464} C_VEL
LIN {X 0,Y 416.184,Z 945.534,A -85,B 0,C 180,E1 17865.827,E2 17865.827} C_VEL
LIN {X 0,Y 394.457,Z 996.937,A -85,B 0,C 180,E1 17874.448,E2 17874.448} C_VEL
LIN {X 0,Y 379.606,Z 1034.182,A -85,B 0,C 180,E1 17884.553,E2 17884.553} C_VEL
LIN {X 0,Y 372.699,Z 1056.502,A -85,B 0,C 180,E1 17894.665,E2 17894.665} C_VEL
LIN {X 0,Y 371.184,Z 1067.169,A -85,B 0,C 180,E1 17904.139,E2 17904.139} C_VEL
LIN {X 0,Y 371.178,Z 1068.504,A -85,B 0,C 180,E1 17913.514,E2 17913.514} C_VEL
LIN {X 0,Y 372.61,Z 1059.122,A -85,B 0,C 180,E1 17924.134,E2 17924.134} C_VEL
LIN {X 0,Y 379.463,Z 1036.007,A -85,B 0,C 180,E1 17935.41,E2 17935.41} C_VEL
LIN {X 0,Y 395.364,Z 999.032,A -85,B 0,C 180,E1 17945.797,E2 17945.797} C_VEL
LIN {X 0,Y 417.81,Z 949.582,A -85,B 0,C 180,E1 17954.321,E2 17954.321} C_VEL
LIN {X 0,Y 442.081,Z 889.801,A -85,B 0,C 180,E1 17960.709,E2 17960.709} C_VEL
LIN {X 0,Y 463.982,Z 820.195,A -85,B 0,C 180,E1 17965.181,E2 17965.181} C_VEL
LIN {X 0,Y 462.491,Z 808.331,A -85,B 0,C 180,E1 17966.58,E2 17966.58} C_VEL
LIN {X 0,Y 445.364,Z 766.194,A -85,B 0,C 180,E1 17974.349,E2 17974.349} C_VEL
LIN {X 0,Y 428.842,Z 737.093,A -85,B 0,C 180,E1 17982.934,E2 17982.934} C_VEL
LIN {X 0,Y 419.965,Z 723.479,A -85,B 0,C 180,E1 17990.224,E2 17990.224} C_VEL
LIN {X 0,Y 416.825,Z 717.834,A -85,B 0,C 180,E1 17995.801,E2 17995.801} C_VEL
LIN {X 0,Y 418.516,Z 720.572,A -85,B 0,C 180,E1 18004.91,E2 18004.91} C_VEL
LIN {X 0,Y 427.02,Z 733.792,A -85,B 0,C 180,E1 18013.008,E2 18013.008} C_VEL
LIN {X 0,Y 443.078,Z 761.667,A -85,B 0,C 180,E1 18021.849,E2 18021.849} C_VEL
LIN {X 0,Y 459.529,Z 800.978,A -85,B 0,C 180,E1 18029.539,E2 18029.539} C_VEL
LIN {X 0,Y 463.445,Z 819.258,A -85,B 0,C 180,E1 18032.081,E2 18032.081} C_VEL
LIN {X 0,Y 441.993,Z 886.315,A -85,B 0,C 180,E1 18036.499,E2 18036.499} C_VEL
LIN {X 0,Y 417.404,Z 946.115,A -85,B 0,C 180,E1 18043.018,E2 18043.018} C_VEL
LIN {X 0,Y 394.484,Z 996.004,A -85,B 0,C 180,E1 18051.955,E2 18051.955} C_VEL
LIN {X 0,Y 378.845,Z 1031.988,A -85,B 0,C 180,E1 18062.592,E2 18062.592} C_VEL
LIN {X 0,Y 372.523,Z 1052.532,A -85,B 0,C 180,E1 18073.143,E2 18073.143} C_VEL
LIN {X 0,Y 370.976,Z 1060.583,A -85,B 0,C 180,E1 18081.774,E2 18081.774} C_VEL
LIN {X 0,Y 371.179,Z 1060.794,A -85,B 0,C 180,E1 18091.17,E2 18091.17} C_VEL
LIN {X 0,Y 372.997,Z 1050.359,A -85,B 0,C 180,E1 18101.728,E2 18101.728} C_VEL
LIN {X 0,Y 380.071,Z 1026.571,A -85,B 0,C 180,E1 18112.697,E2 18112.697} C_VEL
LIN {X 0,Y 395.95,Z 987.958,A -85,B 0,C 180,E1 18123.032,E2 18123.032} C_VEL
LIN {X 0,Y 418.062,Z 936.617,A -85,B 0,C 180,E1 18131.45,E2 18131.45} C_VEL
LIN {X 0,Y 441.02,Z 875.471,A -85,B 0,C 180,E1 18137.668,E2 18137.668} C_VEL
LIN {X 0,Y 458.448,Z 813.417,A -85,B 0,C 180,E1 18141.644,E2 18141.644} C_VEL
LIN {X 0,Y 442.061,Z 768.035,A -85,B 0,C 180,E1 18148.66,E2 18148.66} C_VEL
LIN {X 0,Y 421.9,Z 730.745,A -85,B 0,C 180,E1 18157.094,E2 18157.094} C_VEL
LIN {X 0,Y 406.516,Z 708.089,A -85,B 0,C 180,E1 18165.899,E2 18165.899} C_VEL
LIN {X 0,Y 401.164,Z 700.998,A -85,B 0,C 180,E1 18171.045,E2 18171.045} C_VEL
LIN {X 0,Y 398.624,Z 695.252,A -85,B 0,C 180,E1 18179.342,E2 18179.342} C_VEL
LIN {X 0,Y 404.74,Z 705.897,A -85,B 0,C 180,E1 18189.466,E2 18189.466} C_VEL
LIN {X 0,Y 417.748,Z 724.04,A -85,B 0,C 180,E1 18197.602,E2 18197.602} C_VEL
LIN {X 0,Y 428.327,Z 740.919,A -85,B 0,C 180,E1 18202.421,E2 18202.421} C_VEL
LIN {X 0,Y 434.464,Z 764.54,A -85,B 0,C 180,E1 18205.87,E2 18205.87} C_VEL
LIN {X 0,Y 451.968,Z 809.634,A -85,B 0,C 180,E1 18213.385,E2 18213.385} C_VEL
LIN {X 0,Y 453.333,Z 821.009,A -85,B 0,C 180,E1 18214.662,E2 18214.662} C_VEL
LIN {X 0,Y 432.644,Z 888.188,A -85,B 0,C 180,E1 18218.997,E2 18218.997} C_VEL
LIN {X 0,Y 409.182,Z 947.783,A -85,B 0,C 180,E1 18225.352,E2 18225.352} C_VEL
LIN {X 0,Y 386.804,Z 998.782,A -85,B 0,C 180,E1 18234.165,E2 18234.165} C_VEL
LIN {X 0,Y 371.476,Z 1035.746,A -85,B 0,C 180,E1 18244.62,E2 18244.62} C_VEL
LIN {X 0,Y 364.451,Z 1058.331,A -85,B 0,C 180,E1 18255.544,E2 18255.544} C_VEL
LIN {X 0,Y 363.028,Z 1068.223,A -85,B 0,C 180,E1 18266.408,E2 18266.408} C_VEL
LIN {X 0,Y 363.222,Z 1067.393,A -85,B 0,C 180,E1 18275.992,E2 18275.992} C_VEL
LIN {X 0,Y 365.296,Z 1055.924,A -85,B 0,C 180,E1 18286.525,E2 18286.525} C_VEL
LIN {X 0,Y 374.105,Z 1030.81,A -85,B 0,C 180,E1 18297.785,E2 18297.785} C_VEL
LIN {X 0,Y 392.398,Z 991.135,A -85,B 0,C 180,E1 18308.194,E2 18308.194} C_VEL
LIN {X 0,Y 417.13,Z 938.129,A -85,B 0,C 180,E1 18316.642,E2 18316.642} C_VEL
LIN {X 0,Y 442.336,Z 875.697,A -85,B 0,C 180,E1 18322.648,E2 18322.648} C_VEL
LIN {X 0,Y 459.165,Z 818.283,A -85,B 0,C 180,E1 18326.287,E2 18326.287} C_VEL
LIN {X 0,Y 443.535,Z 776.198,A -85,B 0,C 180,E1 18333.972,E2 18333.972} C_VEL
LIN {X 0,Y 427.484,Z 745.573,A -85,B 0,C 180,E1 18342.701,E2 18342.701} C_VEL
LIN {X 0,Y 418.146,Z 730.97,A -85,B 0,C 180,E1 18350.576,E2 18350.576} C_VEL
LIN {X 0,Y 415.559,Z 725.719,A -85,B 0,C 180,E1 18355.788,E2 18355.788} C_VEL
LIN {X 0,Y 417.007,Z 728.424,A -85,B 0,C 180,E1 18364.809,E2 18364.809} C_VEL
LIN {X 0,Y 425.209,Z 741.796,A -85,B 0,C 180,E1 18372.934,E2 18372.934} C_VEL
LIN {X 0,Y 440.005,Z 768.956,A -85,B 0,C 180,E1 18381.61,E2 18381.61} C_VEL
LIN {X 0,Y 455.078,Z 806.929,A -85,B 0,C 180,E1 18389.171,E2 18389.171} C_VEL
LIN {X 0,Y 457.927,Z 823.345,A -85,B 0,C 180,E1 18391.443,E2 18391.443} C_VEL
LIN {X 0,Y 435.797,Z 889.523,A -85,B 0,C 180,E1 18395.915,E2 18395.915} C_VEL
LIN {X 0,Y 410.873,Z 947.791,A -85,B 0,C 180,E1 18402.426,E2 18402.426} C_VEL
LIN {X 0,Y 387.643,Z 996.512,A -85,B 0,C 180,E1 18411.335,E2 18411.335} C_VEL
LIN {X 0,Y 371.494,Z 1031.963,A -85,B 0,C 180,E1 18422.003,E2 18422.003} C_VEL
LIN {X 0,Y 364.64,Z 1052.558,A -85,B 0,C 180,E1 18432.767,E2 18432.767} C_VEL
LIN {X 0,Y 362.875,Z 1061.599,A -85,B 0,C 180,E1 18444.003,E2 18444.003} C_VEL
LIN {X 0,Y 363.519,Z 1059.573,A -85,B 0,C 180,E1 18453.587,E2 18453.587} C_VEL
LIN {X 0,Y 365.868,Z 1046.64,A -85,B 0,C 180,E1 18464.399,E2 18464.399} C_VEL
LIN {X 0,Y 375.664,Z 1019.188,A -85,B 0,C 180,E1 18475.717,E2 18475.717} C_VEL
LIN {X 0,Y 393.927,Z 977.687,A -85,B 0,C 180,E1 18485.798,E2 18485.798} C_VEL
LIN {X 0,Y 417.456,Z 923.772,A -85,B 0,C 180,E1 18493.823,E2 18493.823} C_VEL
LIN {X 0,Y 440.246,Z 862.304,A -85,B 0,C 180,E1 18499.458,E2 18499.458} C_VEL
LIN {X 0,Y 452.512,Z 815.699,A -85,B 0,C 180,E1 18502.455,E2 18502.455} C_VEL
LIN {X 0,Y 437.114,Z 771.875,A -85,B 0,C 180,E1 18509.523,E2 18509.523} C_VEL
LIN {X 0,Y 418.21,Z 735.883,A -85,B 0,C 180,E1 18518.043,E2 18518.043} C_VEL
LIN {X 0,Y 404.051,Z 714.549,A -85,B 0,C 180,E1 18526.902,E2 18526.902} C_VEL
LIN {X 0,Y 399.485,Z 708.404,A -85,B 0,C 180,E1 18531.833,E2 18531.833} C_VEL
LIN {X 0,Y 397.633,Z 703.317,A -85,B 0,C 180,E1 18539.34,E2 18539.34} C_VEL
LIN {X 0,Y 403.418,Z 713.825,A -85,B 0,C 180,E1 18549.361,E2 18549.361} C_VEL
LIN {X 0,Y 416.893,Z 733.935,A -85,B 0,C 180,E1 18558.05,E2 18558.05} C_VEL
LIN {X 0,Y 434.464,Z 764.54,A -85,B 0,C 180,E1 18565.87,E2 18565.87} C_VEL
LIN {X 0,Y 438.91,Z 790.206,A -85,B 0,C 180,E1 18569.068,E2 18569.068} C_VEL
LIN {X 0,Y 447.879,Z 823.601,A -85,B 0,C 180,E1 18573.952,E2 18573.952} C_VEL
LIN {X 0,Y 426.5,Z 890.659,A -85,B 0,C 180,E1 18578.379,E2 18578.379} C_VEL
LIN {X 0,Y 402.14,Z 950.232,A -85,B 0,C 180,E1 18584.89,E2 18584.89} C_VEL
LIN {X 0,Y 379.894,Z 998.974,A -85,B 0,C 180,E1 18593.515,E2 18593.515} C_VEL
LIN {X 0,Y 364.02,Z 1035.594,A -85,B 0,C 180,E1 18604.062,E2 18604.062} C_VEL
LIN {X 0,Y 356.544,Z 1058.208,A -85,B 0,C 180,E1 18615.216,E2 18615.216} C_VEL
LIN {X 0,Y 355.172,Z 1066.975,A -85,B 0,C 180,E1 18623.873,E2 18623.873} C_VEL
LIN {X 0,Y 355.164,Z 1068.37,A -85,B 0,C 180,E1 18633.673,E2 18633.673} C_VEL
LIN {X 0,Y 356.768,Z 1059.033,A -85,B 0,C 180,E1 18644.776,E2 18644.776} C_VEL
LIN {X 0,Y 364.751,Z 1035.6,A -85,B 0,C 180,E1 18656.682,E2 18656.682} C_VEL
LIN {X 0,Y 382.633,Z 997.889,A -85,B 0,C 180,E1 18667.519,E2 18667.519} C_VEL
LIN {X 0,Y 407.158,Z 947.57,A -85,B 0,C 180,E1 18676.252,E2 18676.252} C_VEL
LIN {X 0,Y 433.098,Z 887.426,A -85,B 0,C 180,E1 18682.596,E2 18682.596} C_VEL
LIN {X 0,Y 453.98,Z 822.708,A -85,B 0,C 180,E1 18686.856,E2 18686.856} C_VEL
LIN {X 0,Y 439.367,Z 781.273,A -85,B 0,C 180,E1 18694.668,E2 18694.668} C_VEL
LIN {X 0,Y 424.532,Z 752.258,A -85,B 0,C 180,E1 18703.318,E2 18703.318} C_VEL
LIN {X 0,Y 416.427,Z 738.638,A -85,B 0,C 180,E1 18710.802,E2 18710.802} C_VEL
LIN {X 0,Y 414.055,Z 733.555,A -85,B 0,C 180,E1 18715.773,E2 18715.773} C_VEL
LIN {X 0,Y 415.396,Z 736.273,A -85,B 0,C 180,E1 18724.693,E2 18724.693} C_VEL
LIN {X 0,Y 423.051,Z 749.517,A -85,B 0,C 180,E1 18732.803,E2 18732.803} C_VEL
LIN {X 0,Y 436.905,Z 776.255,A -85,B 0,C 180,E1 18741.37,E2 18741.37} C_VEL
LIN {X 0,Y 450.709,Z 813.602,A -85,B 0,C 180,E1 18748.929,E2 18748.929} C_VEL
LIN {X 0,Y 452.512,Z 827.2,A -85,B 0,C 180,E1 18750.78,E2 18750.78} C_VEL
LIN {X 0,Y 429.606,Z 892.687,A -85,B 0,C 180,E1 18755.327,E2 18755.327} C_VEL
LIN {X 0,Y 403.492,Z 951.179,A -85,B 0,C 180,E1 18762.076,E2 18762.076} C_VEL
LIN {X 0,Y 379.611,Z 999.158,A -85,B 0,C 180,E1 18771.19,E2 18771.19} C_VEL
LIN {X 0,Y 363.444,Z 1033.479,A -85,B 0,C 180,E1 18782.005,E2 18782.005} C_VEL
LIN {X 0,Y 356.516,Z 1053.637,A -85,B 0,C 180,E1 18793.221,E2 18793.221} C_VEL
LIN {X 0,Y 354.865,Z 1061.671,A -85,B 0,C 180,E1 18803.867,E2 18803.867} C_VEL
LIN {X 0,Y 355.53,Z 1059.68,A -85,B 0,C 180,E1 18813.668,E2 18813.668} C_VEL
LIN {X 0,Y 358.026,Z 1046.797,A -85,B 0,C 180,E1 18824.721,E2 18824.721} C_VEL
LIN {X 0,Y 368.325,Z 1019.398,A -85,B 0,C 180,E1 18836.268,E2 18836.268} C_VEL
LIN {X 0,Y 387.15,Z 978.292,A -85,B 0,C 180,E1 18846.444,E2 18846.444} C_VEL
LIN {X 0,Y 411.637,Z 924.129,A -85,B 0,C 180,E1 18854.605,E2 18854.605} C_VEL
LIN {X 0,Y 435.073,Z 862.78,A -85,B 0,C 180,E1 18860.26,E2 18860.26} C_VEL
LIN {X 0,Y 447.061,Z 819.664,A -85,B 0,C 180,E1 18863.05,E2 18863.05} C_VEL
LIN {X 0,Y 432.605,Z 776.644,A -85,B 0,C 180,E1 18870.225,E2 18870.225} C_VEL
LIN {X 0,Y 415.124,Z 742.326,A -85,B 0,C 180,E1 18878.667,E2 18878.667} C_VEL
LIN {X 0,Y 402.19,Z 721.602,A -85,B 0,C 180,E1 18887.486,E2 18887.486} C_VEL
LIN {X 0,Y 396.554,Z 710.744,A -85,B 0,C 180,E1 18897.83,E2 18897.83} C_VEL
LIN {X 0,Y 401.886,Z 721.378,A -85,B 0,C 180,E1 18909.055,E2 18909.055} C_VEL
LIN {X 0,Y 414.858,Z 741.589,A -85,B 0,C 180,E1 18917.867,E2 18917.867} C_VEL
LIN {X 0,Y 433.501,Z 776.785,A -85,B 0,C 180,E1 18926.627,E2 18926.627} C_VEL
LIN {X 0,Y 438.91,Z 790.206,A -85,B 0,C 180,E1 18929.068,E2 18929.068} C_VEL
LIN {X 0,Y 441.257,Z 817.253,A -85,B 0,C 180,E1 18932.079,E2 18932.079} C_VEL
LIN {X 0,Y 442.302,Z 827.05,A -85,B 0,C 180,E1 18933.275,E2 18933.275} C_VEL
LIN {X 0,Y 420.71,Z 892.27,A -85,B 0,C 180,E1 18937.669,E2 18937.669} C_VEL
LIN {X 0,Y 395.521,Z 951.795,A -85,B 0,C 180,E1 18944.292,E2 18944.292} C_VEL
LIN {X 0,Y 371.966,Z 1001.243,A -85,B 0,C 180,E1 18953.336,E2 18953.336} C_VEL
LIN {X 0,Y 355.197,Z 1038.548,A -85,B 0,C 180,E1 18964.728,E2 18964.728} C_VEL
LIN {X 0,Y 348.307,Z 1059.715,A -85,B 0,C 180,E1 18976.146,E2 18976.146} C_VEL
LIN {X 0,Y 347.034,Z 1068.044,A -85,B 0,C 180,E1 18986.242,E2 18986.242} C_VEL
LIN {X 0,Y 347.217,Z 1067.259,A -85,B 0,C 180,E1 18996.269,E2 18996.269} C_VEL
LIN {X 0,Y 349.682,Z 1055.497,A -85,B 0,C 180,E1 19007.525,E2 19007.525} C_VEL
LIN {X 0,Y 360.136,Z 1029.598,A -85,B 0,C 180,E1 19019.446,E2 19019.446} C_VEL
LIN {X 0,Y 381.034,Z 988.582,A -85,B 0,C 180,E1 19030.294,E2 19030.294} C_VEL
LIN {X 0,Y 407.471,Z 935.249,A -85,B 0,C 180,E1 19038.702,E2 19038.702} C_VEL
LIN {X 0,Y 433.888,Z 872.779,A -85,B 0,C 180,E1 19044.61,E2 19044.61} C_VEL
LIN {X 0,Y 448.483,Z 825.919,A -85,B 0,C 180,E1 19047.645,E2 19047.645} C_VEL
LIN {X 0,Y 434.896,Z 785.909,A -85,B 0,C 180,E1 19055.492,E2 19055.492} C_VEL
LIN {X 0,Y 421.372,Z 758.351,A -85,B 0,C 180,E1 19064.154,E2 19064.154} C_VEL
LIN {X 0,Y 414.113,Z 745.412,A -85,B 0,C 180,E1 19071.679,E2 19071.679} C_VEL
LIN {X 0,Y 412.26,Z 741.278,A -85,B 0,C 180,E1 19076.811,E2 19076.811} C_VEL
LIN {X 0,Y 413.642,Z 744.087,A -85,B 0,C 180,E1 19084.581,E2 19084.581} C_VEL
LIN {X 0,Y 420.893,Z 757.249,A -85,B 0,C 180,E1 19092.671,E2 19092.671} C_VEL
LIN {X 0,Y 434.208,Z 784.829,A -85,B 0,C 180,E1 19101.509,E2 19101.509} C_VEL
LIN {X 0,Y 446.954,Z 822.747,A -85,B 0,C 180,E1 19109.132,E2 19109.132} C_VEL
LIN {X 0,Y 446.506,Z 832.513,A -85,B 0,C 180,E1 19110.187,E2 19110.187} C_VEL
LIN {X 0,Y 422.419,Z 898.183,A -85,B 0,C 180,E1 19114.949,E2 19114.949} C_VEL
LIN {X 0,Y 395.414,Z 956.028,A -85,B 0,C 180,E1 19121.937,E2 19121.937} C_VEL
LIN {X 0,Y 370.85,Z 1003.327,A -85,B 0,C 180,E1 19131.422,E2 19131.422} C_VEL
LIN {X 0,Y 354.714,Z 1036.432,A -85,B 0,C 180,E1 19142.64,E2 19142.64} C_VEL
LIN {X 0,Y 348.442,Z 1054.56,A -85,B 0,C 180,E1 19153.567,E2 19153.567} C_VEL
LIN {X 0,Y 346.857,Z 1061.744,A -85,B 0,C 180,E1 19163.725,E2 19163.725} C_VEL
LIN {X 0,Y 347.525,Z 1059.787,A -85,B 0,C 180,E1 19173.752,E2 19173.752} C_VEL
LIN {X 0,Y 350.186,Z 1046.953,A -85,B 0,C 180,E1 19185.059,E2 19185.059} C_VEL
LIN {X 0,Y 361.029,Z 1019.607,A -85,B 0,C 180,E1 19196.841,E2 19196.841} C_VEL
LIN {X 0,Y 381.167,Z 977.434,A -85,B 0,C 180,E1 19207.392,E2 19207.392} C_VEL
LIN {X 0,Y 406.365,Z 923.432,A -85,B 0,C 180,E1 19215.534,E2 19215.534} C_VEL
LIN {X 0,Y 430.52,Z 861.715,A -85,B 0,C 180,E1 19221.196,E2 19221.196} C_VEL
LIN {X 0,Y 441.404,Z 822.371,A -85,B 0,C 180,E1 19223.835,E2 19223.835} C_VEL
LIN {X 0,Y 427.167,Z 779.331,A -85,B 0,C 180,E1 19231.361,E2 19231.361} C_VEL
LIN {X 0,Y 410.838,Z 746.516,A -85,B 0,C 180,E1 19239.97,E2 19239.97} C_VEL
LIN {X 0,Y 398.897,Z 725.577,A -85,B 0,C 180,E1 19249.6,E2 19249.6} C_VEL
LIN {X 0,Y 395.325,Z 719.397,A -85,B 0,C 180,E1 19259.336,E2 19259.336} C_VEL
LIN {X 0,Y 400.654,Z 729.823,A -85,B 0,C 180,E1 19269.289,E2 19269.289} C_VEL
LIN {X 0,Y 413.714,Z 751.008,A -85,B 0,C 180,E1 19278.332,E2 19278.332} C_VEL
LIN {X 0,Y 430.928,Z 786.121,A -85,B 0,C 180,E1 19286.843,E2 19286.843} C_VEL
LIN {X 0,Y 441.257,Z 817.253,A -85,B 0,C 180,E1 19292.079,E2 19292.079} C_VEL
LIN {X 0,Y 436.423,Z 833.37,A -85,B 0,C 180,E1 19292.83,E2 19292.83} C_VEL
LIN {X 0,Y 434.143,Z 838.966,A -85,B 0,C 180,E1 19293.04,E2 19293.04} C_VEL
LIN {X 0,Y 410.178,Z 905.546,A -85,B 0,C 180,E1 19298.01,E2 19298.01} C_VEL
LIN {X 0,Y 383.95,Z 963.582,A -85,B 0,C 180,E1 19305.247,E2 19305.247} C_VEL
LIN {X 0,Y 360.338,Z 1010.838,A -85,B 0,C 180,E1 19315.014,E2 19315.014} C_VEL
LIN {X 0,Y 345.596,Z 1043.542,A -85,B 0,C 180,E1 19326.372,E2 19326.372} C_VEL
LIN {X 0,Y 339.874,Z 1062.604,A -85,B 0,C 180,E1 19338.418,E2 19338.418} C_VEL
LIN {X 0,Y 339.085,Z 1068.588,A -85,B 0,C 180,E1 19348.719,E2 19348.719} C_VEL
LIN {X 0,Y 339.514,Z 1065.517,A -85,B 0,C 180,E1 19358.994,E2 19358.994} C_VEL
LIN {X 0,Y 344.124,Z 1049.802,A -85,B 0,C 180,E1 19371.319,E2 19371.319} C_VEL
LIN {X 0,Y 358.891,Z 1018.601,A -85,B 0,C 180,E1 19383.682,E2 19383.682} C_VEL
LIN {X 0,Y 382.669,Z 973.831,A -85,B 0,C 180,E1 19393.907,E2 19393.907} C_VEL
LIN {X 0,Y 409.761,Z 919.149,A -85,B 0,C 180,E1 19401.428,E2 19401.428} C_VEL
LIN {X 0,Y 436.201,Z 853.966,A -85,B 0,C 180,E1 19406.774,E2 19406.774} C_VEL
LIN {X 0,Y 443.445,Z 830.457,A -85,B 0,C 180,E1 19408.223,E2 19408.223} C_VEL
LIN {X 0,Y 430.927,Z 791.573,A -85,B 0,C 180,E1 19416.082,E2 19416.082} C_VEL
LIN {X 0,Y 418.414,Z 764.842,A -85,B 0,C 180,E1 19424.762,E2 19424.762} C_VEL
LIN {X 0,Y 411.332,Z 749.557,A -85,B 0,C 180,E1 19434.153,E2 19434.153} C_VEL
LIN {X 0,Y 411.646,Z 751.626,A -85,B 0,C 180,E1 19444.338,E2 19444.338} C_VEL
LIN {X 0,Y 418.586,Z 765.224,A -85,B 0,C 180,E1 19452.676,E2 19452.676} C_VEL
LIN {X 0,Y 430.735,Z 791.655,A -85,B 0,C 180,E1 19461.203,E2 19461.203} C_VEL
LIN {X 0,Y 442.485,Z 829.79,A -85,B 0,C 180,E1 19468.984,E2 19468.984} C_VEL
LIN {X 0,Y 417.591,Z 898.215,A -85,B 0,C 180,E1 19474.04,E2 19474.04} C_VEL
LIN {X 0,Y 389.911,Z 955.745,A -85,B 0,C 180,E1 19480.997,E2 19480.997} C_VEL
LIN {X 0,Y 364.789,Z 1002.423,A -85,B 0,C 180,E1 19490.394,E2 19490.394} C_VEL
LIN {X 0,Y 347.307,Z 1036.426,A -85,B 0,C 180,E1 19502.008,E2 19502.008} C_VEL
LIN {X 0,Y 340.544,Z 1054.719,A -85,B 0,C 180,E1 19513.287,E2 19513.287} C_VEL
LIN {X 0,Y 338.866,Z 1061.816,A -85,B 0,C 180,E1 19523.576,E2 19523.576} C_VEL
LIN {X 0,Y 339.537,Z 1059.893,A -85,B 0,C 180,E1 19533.841,E2 19533.841} C_VEL
LIN {X 0,Y 342.364,Z 1047.108,A -85,B 0,C 180,E1 19545.411,E2 19545.411} C_VEL
LIN {X 0,Y 353.795,Z 1019.814,A -85,B 0,C 180,E1 19557.435,E2 19557.435} C_VEL
LIN {X 0,Y 374.382,Z 978.358,A -85,B 0,C 180,E1 19568.022,E2 19568.022} C_VEL
LIN {X 0,Y 400.751,Z 923.777,A -85,B 0,C 180,E1 19576.358,E2 19576.358} C_VEL
LIN {X 0,Y 426.093,Z 860.659,A -85,B 0,C 180,E1 19582.15,E2 19582.15} C_VEL
LIN {X 0,Y 436.198,Z 826.868,A -85,B 0,C 180,E1 19584.377,E2 19584.377} C_VEL
LIN {X 0,Y 423.166,Z 785.344,A -85,B 0,C 180,E1 19591.827,E2 19591.827} C_VEL
LIN {X 0,Y 407.683,Z 752.407,A -85,B 0,C 180,E1 19600.692,E2 19600.692} C_VEL
LIN {X 0,Y 396.883,Z 733.193,A -85,B 0,C 180,E1 19610.115,E2 19610.115} C_VEL
LIN {X 0,Y 393.965,Z 727.346,A -85,B 0,C 180,E1 19619.334,E2 19619.334} C_VEL
LIN {X 0,Y 398.916,Z 737.566,A -85,B 0,C 180,E1 19629.123,E2 19629.123} C_VEL
LIN {X 0,Y 411.188,Z 758.517,A -85,B 0,C 180,E1 19638.096,E2 19638.096} C_VEL
LIN {X 0,Y 427.341,Z 793.602,A -85,B 0,C 180,E1 19646.666,E2 19646.666} C_VEL
LIN {X 0,Y 437.049,Z 829.544,A -85,B 0,C 180,E1 19652.533,E2 19652.533} C_VEL
LIN {X 0,Y 434.143,Z 838.966,A -85,B 0,C 180,E1 19653.04,E2 19653.04} C_VEL
LIN {X 0,Y 418.968,Z 869.991,A -85,B 0,C 180,E1 19654.119,E2 19654.119} C_VEL
LIN {X 0,Y 392.445,Z 933.547,A -85,B 0,C 180,E1 19660.166,E2 19660.166} C_VEL
LIN {X 0,Y 366.244,Z 986.554,A -85,B 0,C 180,E1 19668.588,E2 19668.588} C_VEL
LIN {X 0,Y 345.114,Z 1028.124,A -85,B 0,C 180,E1 19679.649,E2 19679.649} C_VEL
LIN {X 0,Y 334.344,Z 1053.932,A -85,B 0,C 180,E1 19691.49,E2 19691.49} C_VEL
LIN {X 0,Y 331.184,Z 1066.681,A -85,B 0,C 180,E1 19703.428,E2 19703.428} C_VEL
LIN {X 0,Y 331.146,Z 1068.171,A -85,B 0,C 180,E1 19713.939,E2 19713.939} C_VEL
LIN {X 0,Y 333.078,Z 1058.904,A -85,B 0,C 180,E1 19725.853,E2 19725.853} C_VEL
LIN {X 0,Y 342.51,Z 1035.893,A -85,B 0,C 180,E1 19738.421,E2 19738.421} C_VEL
LIN {X 0,Y 363.012,Z 998.428,A -85,B 0,C 180,E1 19749.823,E2 19749.823} C_VEL
LIN {X 0,Y 390.418,Z 948.085,A -85,B 0,C 180,E1 19758.844,E2 19758.844} C_VEL
LIN {X 0,Y 418.783,Z 887.936,A -85,B 0,C 180,E1 19765.253,E2 19765.253} C_VEL
LIN {X 0,Y 438.138,Z 834.135,A -85,B 0,C 180,E1 19768.945,E2 19768.945} C_VEL
LIN {X 0,Y 426.915,Z 797.156,A -85,B 0,C 180,E1 19776.709,E2 19776.709} C_VEL
LIN {X 0,Y 415.157,Z 770.479,A -85,B 0,C 180,E1 19785.673,E2 19785.673} C_VEL
LIN {X 0,Y 409.006,Z 757.099,A -85,B 0,C 180,E1 19795.187,E2 19795.187} C_VEL
LIN {X 0,Y 409.7,Z 759.461,A -85,B 0,C 180,E1 19804.293,E2 19804.293} C_VEL
LIN {X 0,Y 416.097,Z 772.846,A -85,B 0,C 180,E1 19812.552,E2 19812.552} C_VEL
LIN {X 0,Y 427.339,Z 799.231,A -85,B 0,C 180,E1 19821.11,E2 19821.11} C_VEL
LIN {X 0,Y 437.381,Z 834.45,A -85,B 0,C 180,E1 19828.439,E2 19828.439} C_VEL
LIN {X 0,Y 411.791,Z 900.73,A -85,B 0,C 180,E1 19833.348,E2 19833.348} C_VEL
LIN {X 0,Y 382.822,Z 958.72,A -85,B 0,C 180,E1 19840.538,E2 19840.538} C_VEL
LIN {X 0,Y 357.198,Z 1004.292,A -85,B 0,C 180,E1 19850.045,E2 19850.045} C_VEL
LIN {X 0,Y 339.251,Z 1037.755,A -85,B 0,C 180,E1 19862.008,E2 19862.008} C_VEL
LIN {X 0,Y 332.244,Z 1056.203,A -85,B 0,C 180,E1 19874.27,E2 19874.27} C_VEL
LIN {X 0,Y 331.046,Z 1062.224,A -85,B 0,C 180,E1 19886.059,E2 19886.059} C_VEL
LIN {X 0,Y 331.668,Z 1058.204,A -85,B 0,C 180,E1 19896.563,E2 19896.563} C_VEL
LIN {X 0,Y 337.13,Z 1041.175,A -85,B 0,C 180,E1 19909.213,E2 19909.213} C_VEL
LIN {X 0,Y 352.338,Z 1009.057,A -85,B 0,C 180,E1 19921.455,E2 19921.455} C_VEL
LIN {X 0,Y 375.46,Z 964.532,A -85,B 0,C 180,E1 19931.403,E2 19931.403} C_VEL
LIN {X 0,Y 402.662,Z 907.519,A -85,B 0,C 180,E1 19939.056,E2 19939.056} C_VEL
LIN {X 0,Y 427.588,Z 842.497,A -85,B 0,C 180,E1 19944.232,E2 19944.232} C_VEL
LIN {X 0,Y 430.341,Z 828.421,A -85,B 0,C 180,E1 19945.377,E2 19945.377} C_VEL
LIN {X 0,Y 417.349,Z 786.841,A -85,B 0,C 180,E1 19953.322,E2 19953.322} C_VEL
LIN {X 0,Y 403.814,Z 757.599,A -85,B 0,C 180,E1 19961.879,E2 19961.879} C_VEL
LIN {X 0,Y 394.915,Z 740.751,A -85,B 0,C 180,E1 19970.623,E2 19970.623} C_VEL
LIN {X 0,Y 392.435,Z 735.29,A -85,B 0,C 180,E1 19979.332,E2 19979.332} C_VEL
LIN {X 0,Y 397.294,Z 745.659,A -85,B 0,C 180,E1 19989.229,E2 19989.229} C_VEL
LIN {X 0,Y 408.825,Z 766.91,A -85,B 0,C 180,E1 19998.133,E2 19998.133} C_VEL
LIN {X 0,Y 423.826,Z 801.542,A -85,B 0,C 180,E1 20006.617,E2 20006.617} C_VEL
LIN {X 0,Y 431.663,Z 832.563,A -85,B 0,C 180,E1 20011.802,E2 20011.802} C_VEL
LIN {X 0,Y 418.968,Z 869.991,A -85,B 0,C 180,E1 20014.119,E2 20014.119} C_VEL
LIN {X 0,Y 402.564,Z 899.534,A -85,B 0,C 180,E1 20015.648,E2 20015.648} C_VEL
LIN {X 0,Y 374.472,Z 958.819,A -85,B 0,C 180,E1 20022.781,E2 20022.781} C_VEL
LIN {X 0,Y 348.706,Z 1006.95,A -85,B 0,C 180,E1 20032.497,E2 20032.497} C_VEL
LIN {X 0,Y 331.466,Z 1041.193,A -85,B 0,C 180,E1 20044.24,E2 20044.24} C_VEL
LIN {X 0,Y 324.268,Z 1060.954,A -85,B 0,C 180,E1 20056.479,E2 20056.479} C_VEL
LIN {X 0,Y 323.033,Z 1067.775,A -85,B 0,C 180,E1 20065.963,E2 20065.963} C_VEL
LIN {X 0,Y 323.137,Z 1068.104,A -85,B 0,C 180,E1 20074.037,E2 20074.037} C_VEL
LIN {X 0,Y 325.112,Z 1059.243,A -85,B 0,C 180,E1 20085.915,E2 20085.915} C_VEL
LIN {X 0,Y 334.429,Z 1037.425,A -85,B 0,C 180,E1 20098.432,E2 20098.432} C_VEL
LIN {X 0,Y 355.059,Z 1001.171,A -85,B 0,C 180,E1 20110.016,E2 20110.016} C_VEL
LIN {X 0,Y 383.534,Z 951.124,A -85,B 0,C 180,E1 20119.365,E2 20119.365} C_VEL
LIN {X 0,Y 412.38,Z 892.389,A -85,B 0,C 180,E1 20125.831,E2 20125.831} C_VEL
LIN {X 0,Y 432.811,Z 837.682,A -85,B 0,C 180,E1 20129.71,E2 20129.71} C_VEL
LIN {X 0,Y 422.148,Z 800.948,A -85,B 0,C 180,E1 20137.796,E2 20137.796} C_VEL
LIN {X 0,Y 411.672,Z 776.13,A -85,B 0,C 180,E1 20146.814,E2 20146.814} C_VEL
LIN {X 0,Y 406.731,Z 764.699,A -85,B 0,C 180,E1 20155.697,E2 20155.697} C_VEL
LIN {X 0,Y 407.384,Z 767.038,A -85,B 0,C 180,E1 20164.116,E2 20164.116} C_VEL
LIN {X 0,Y 413.364,Z 780.252,A -85,B 0,C 180,E1 20172.367,E2 20172.367} C_VEL
LIN {X 0,Y 423.799,Z 806.561,A -85,B 0,C 180,E1 20180.962,E2 20180.962} C_VEL
LIN {X 0,Y 432.164,Z 838.332,A -85,B 0,C 180,E1 20187.74,E2 20187.74} C_VEL
LIN {X 0,Y 405.585,Z 904.253,A -85,B 0,C 180,E1 20192.728,E2 20192.728} C_VEL
LIN {X 0,Y 375.721,Z 961.622,A -85,B 0,C 180,E1 20200.078,E2 20200.078} C_VEL
LIN {X 0,Y 349.052,Z 1006.972,A -85,B 0,C 180,E1 20209.944,E2 20209.944} C_VEL
LIN {X 0,Y 331.241,Z 1039.02,A -85,B 0,C 180,E1 20221.977,E2 20221.977} C_VEL
LIN {X 0,Y 324.472,Z 1055.842,A -85,B 0,C 180,E1 20233.42,E2 20233.42} C_VEL
LIN {X 0,Y 323.023,Z 1062.297,A -85,B 0,C 180,E1 20245.961,E2 20245.961} C_VEL
LIN {X 0,Y 323.706,Z 1058.322,A -85,B 0,C 180,E1 20256.725,E2 20256.725} C_VEL
LIN {X 0,Y 329.261,Z 1041.826,A -85,B 0,C 180,E1 20269.434,E2 20269.434} C_VEL
LIN {X 0,Y 344.818,Z 1010.349,A -85,B 0,C 180,E1 20281.851,E2 20281.851} C_VEL
LIN {X 0,Y 368.516,Z 966.457,A -85,B 0,C 180,E1 20291.949,E2 20291.949} C_VEL
LIN {X 0,Y 396.38,Z 910.131,A -85,B 0,C 180,E1 20299.695,E2 20299.695} C_VEL
LIN {X 0,Y 422.287,Z 844.972,A -85,B 0,C 180,E1 20304.994,E2 20304.994} C_VEL
LIN {X 0,Y 425.203,Z 833.583,A -85,B 0,C 180,E1 20305.818,E2 20305.818} C_VEL
LIN {X 0,Y 414.027,Z 794.343,A -85,B 0,C 180,E1 20313.46,E2 20313.46} C_VEL
LIN {X 0,Y 401.147,Z 764.941,A -85,B 0,C 180,E1 20322.121,E2 20322.121} C_VEL
LIN {X 0,Y 392.864,Z 748.388,A -85,B 0,C 180,E1 20330.854,E2 20330.854} C_VEL
LIN {X 0,Y 390.83,Z 743.202,A -85,B 0,C 180,E1 20339.381,E2 20339.381} C_VEL
LIN {X 0,Y 395.492,Z 753.654,A -85,B 0,C 180,E1 20349.342,E2 20349.342} C_VEL
LIN {X 0,Y 407.195,Z 776.708,A -85,B 0,C 180,E1 20358.663,E2 20358.663} C_VEL
LIN {X 0,Y 420.584,Z 810.867,A -85,B 0,C 180,E1 20366.839,E2 20366.839} C_VEL
LIN {X 0,Y 425.686,Z 837.327,A -85,B 0,C 180,E1 20371.157,E2 20371.157} C_VEL
LIN {X 0,Y 402.564,Z 899.534,A -85,B 0,C 180,E1 20375.648,E2 20375.648} C_VEL
LIN {X 0,Y 384.833,Z 927.273,A -85,B 0,C 180,E1 20377.586,E2 20377.586} C_VEL
LIN {X 0,Y 356.463,Z 981.412,A -85,B 0,C 180,E1 20385.857,E2 20385.857} C_VEL
LIN {X 0,Y 332.686,Z 1023.947,A -85,B 0,C 180,E1 20396.843,E2 20396.843} C_VEL
LIN {X 0,Y 319.293,Z 1052.575,A -85,B 0,C 180,E1 20409.86,E2 20409.86} C_VEL
LIN {X 0,Y 315.196,Z 1066.485,A -85,B 0,C 180,E1 20423.093,E2 20423.093} C_VEL
LIN {X 0,Y 315.129,Z 1068.038,A -85,B 0,C 180,E1 20434.14,E2 20434.14} C_VEL
LIN {X 0,Y 317.209,Z 1059.327,A -85,B 0,C 180,E1 20446.209,E2 20446.209} C_VEL
LIN {X 0,Y 327.151,Z 1037.421,A -85,B 0,C 180,E1 20459.124,E2 20459.124} C_VEL
LIN {X 0,Y 349.265,Z 1000.367,A -85,B 0,C 180,E1 20471.109,E2 20471.109} C_VEL
LIN {X 0,Y 378.825,Z 950.074,A -85,B 0,C 180,E1 20480.477,E2 20480.477} C_VEL
LIN {X 0,Y 408.597,Z 890.958,A -85,B 0,C 180,E1 20486.908,E2 20486.908} C_VEL
LIN {X 0,Y 427.585,Z 841.575,A -85,B 0,C 180,E1 20490.44,E2 20490.44} C_VEL
LIN {X 0,Y 418.001,Z 806.357,A -85,B 0,C 180,E1 20498.483,E2 20498.483} C_VEL
LIN {X 0,Y 408.83,Z 783.391,A -85,B 0,C 180,E1 20507.106,E2 20507.106} C_VEL
LIN {X 0,Y 404.524,Z 772.376,A -85,B 0,C 180,E1 20515.673,E2 20515.673} C_VEL
LIN {X 0,Y 405.116,Z 774.808,A -85,B 0,C 180,E1 20524.089,E2 20524.089} C_VEL
LIN {X 0,Y 411.485,Z 789.645,A -85,B 0,C 180,E1 20533.135,E2 20533.135} C_VEL
LIN {X 0,Y 421.364,Z 818.175,A -85,B 0,C 180,E1 20541.899,E2 20541.899} C_VEL
LIN {X 0,Y 426.17,Z 844.627,A -85,B 0,C 180,E1 20547.166,E2 20547.166} C_VEL
LIN {X 0,Y 398.326,Z 909.818,A -85,B 0,C 180,E1 20552.32,E2 20552.32} C_VEL
LIN {X 0,Y 367.676,Z 965.931,A -85,B 0,C 180,E1 20559.849,E2 20559.849} C_VEL
LIN {X 0,Y 340.965,Z 1009.644,A -85,B 0,C 180,E1 20569.843,E2 20569.843} C_VEL
LIN {X 0,Y 323.153,Z 1040.421,A -85,B 0,C 180,E1 20582.013,E2 20582.013} C_VEL
LIN {X 0,Y 316.119,Z 1057.341,A -85,B 0,C 180,E1 20594.702,E2 20594.702} C_VEL
LIN {X 0,Y 315.003,Z 1062.37,A -85,B 0,C 180,E1 20605.858,E2 20605.858} C_VEL
LIN {X 0,Y 315.726,Z 1058.44,A -85,B 0,C 180,E1 20616.896,E2 20616.896} C_VEL
LIN {X 0,Y 321.715,Z 1041.71,A -85,B 0,C 180,E1 20630.062,E2 20630.062} C_VEL
LIN {X 0,Y 338.426,Z 1009.5,A -85,B 0,C 180,E1 20642.908,E2 20642.908} C_VEL
LIN {X 0,Y 363.24,Z 965.394,A -85,B 0,C 180,E1 20653.048,E2 20653.048} C_VEL
LIN {X 0,Y 391.748,Z 909.311,A -85,B 0,C 180,E1 20660.728,E2 20660.728} C_VEL
LIN {X 0,Y 418.217,Z 844.155,A -85,B 0,C 180,E1 20665.979,E2 20665.979} C_VEL
LIN {X 0,Y 419.301,Z 834.619,A -85,B 0,C 180,E1 20666.984,E2 20666.984} C_VEL
LIN {X 0,Y 408.339,Z 795.874,A -85,B 0,C 180,E1 20675.043,E2 20675.043} C_VEL
LIN {X 0,Y 396.418,Z 767.737,A -85,B 0,C 180,E1 20684.194,E2 20684.194} C_VEL
LIN {X 0,Y 390.253,Z 755.527,A -85,B 0,C 180,E1 20691.92,E2 20691.92} C_VEL
LIN {X 0,Y 388.956,Z 751.014,A -85,B 0,C 180,E1 20699.378,E2 20699.378} C_VEL
LIN {X 0,Y 393.479,Z 761.49,A -85,B 0,C 180,E1 20709.32,E2 20709.32} C_VEL
LIN {X 0,Y 404.37,Z 784.583,A -85,B 0,C 180,E1 20718.63,E2 20718.63} C_VEL
LIN {X 0,Y 416.343,Z 817.436,A -85,B 0,C 180,E1 20726.551,E2 20726.551} C_VEL
LIN {X 0,Y 420.37,Z 840.334,A -85,B 0,C 180,E1 20730.402,E2 20730.402} C_VEL
LIN {X 0,Y 394.64,Z 906.303,A -85,B 0,C 180,E1 20735.354,E2 20735.354} C_VEL
LIN {X 0,Y 384.833,Z 927.273,A -85,B 0,C 180,E1 20737.586,E2 20737.586} C_VEL
LIN {X 0,Y 366.289,Z 952.987,A -85,B 0,C 180,E1 20740.021,E2 20740.021} C_VEL
LIN {X 0,Y 338.611,Z 1001.669,A -85,B 0,C 180,E1 20749.508,E2 20749.508} C_VEL
LIN {X 0,Y 317.867,Z 1038.537,A -85,B 0,C 180,E1 20761.89,E2 20761.89} C_VEL
LIN {X 0,Y 308.837,Z 1059.133,A -85,B 0,C 180,E1 20774.333,E2 20774.333} C_VEL
LIN {X 0,Y 307.034,Z 1067.595,A -85,B 0,C 180,E1 20785.752,E2 20785.752} C_VEL
LIN {X 0,Y 307.128,Z 1067.972,A -85,B 0,C 180,E1 20794.248,E2 20794.248} C_VEL
LIN {X 0,Y 309.399,Z 1059.06,A -85,B 0,C 180,E1 20806.839,E2 20806.839} C_VEL
LIN {X 0,Y 320.915,Z 1035.88,A -85,B 0,C 180,E1 20820.529,E2 20820.529} C_VEL
LIN {X 0,Y 344.541,Z 998.121,A -85,B 0,C 180,E1 20832.587,E2 20832.587} C_VEL
LIN {X 0,Y 374.775,Z 948.193,A -85,B 0,C 180,E1 20841.72,E2 20841.72} C_VEL
LIN {X 0,Y 405.835,Z 887.646,A -85,B 0,C 180,E1 20848.15,E2 20848.15} C_VEL
LIN {X 0,Y 422.377,Z 845.148,A -85,B 0,C 180,E1 20851.248,E2 20851.248} C_VEL
LIN {X 0,Y 414.057,Z 812.246,A -85,B 0,C 180,E1 20859.051,E2 20859.051} C_VEL
LIN {X 0,Y 405.385,Z 789.395,A -85,B 0,C 180,E1 20868.093,E2 20868.093} C_VEL
LIN {X 0,Y 402.591,Z 780.263,A -85,B 0,C 180,E1 20874.568,E2 20874.568} C_VEL
LIN {X 0,Y 402.51,Z 781.302,A -85,B 0,C 180,E1 20883.274,E2 20883.274} C_VEL
LIN {X 0,Y 408.356,Z 796.741,A -85,B 0,C 180,E1 20892.862,E2 20892.862} C_VEL
LIN {X 0,Y 417.088,Z 824.021,A -85,B 0,C 180,E1 20901.428,E2 20901.428} C_VEL
LIN {X 0,Y 420.99,Z 848.05,A -85,B 0,C 180,E1 20906.4,E2 20906.4} C_VEL
LIN {X 0,Y 392.227,Z 912.923,A -85,B 0,C 180,E1 20911.644,E2 20911.644} C_VEL
LIN {X 0,Y 360.51,Z 968.901,A -85,B 0,C 180,E1 20919.383,E2 20919.383} C_VEL
LIN {X 0,Y 332.579,Z 1012.859,A -85,B 0,C 180,E1 20929.906,E2 20929.906} C_VEL
LIN {X 0,Y 314.534,Z 1042.979,A -85,B 0,C 180,E1 20942.741,E2 20942.741} C_VEL
LIN {X 0,Y 307.902,Z 1058.587,A -85,B 0,C 180,E1 20955.744,E2 20955.744} C_VEL
LIN {X 0,Y 307.26,Z 1062.259,A -85,B 0,C 180,E1 20968.585,E2 20968.585} C_VEL
LIN {X 0,Y 308.871,Z 1054.747,A -85,B 0,C 180,E1 20981.288,E2 20981.288} C_VEL
LIN {X 0,Y 317.783,Z 1033.703,A -85,B 0,C 180,E1 20994.738,E2 20994.738} C_VEL
LIN {X 0,Y 337.759,Z 998.755,A -85,B 0,C 180,E1 21006.817,E2 21006.817} C_VEL
LIN {X 0,Y 365.859,Z 950.313,A -85,B 0,C 180,E1 21016.496,E2 21016.496} C_VEL
LIN {X 0,Y 395.286,Z 891.059,A -85,B 0,C 180,E1 21023.472,E2 21023.472} C_VEL
LIN {X 0,Y 414.402,Z 840.484,A -85,B 0,C 180,E1 21027.328,E2 21027.328} C_VEL
LIN {X 0,Y 404.598,Z 802.622,A -85,B 0,C 180,E1 21035.338,E2 21035.338} C_VEL
LIN {X 0,Y 393.716,Z 775.001,A -85,B 0,C 180,E1 21044.513,E2 21044.513} C_VEL
LIN {X 0,Y 388.051,Z 763.089,A -85,B 0,C 180,E1 21052.156,E2 21052.156} C_VEL
LIN {X 0,Y 387.055,Z 759.021,A -85,B 0,C 180,E1 21059.533,E2 21059.533} C_VEL
LIN {X 0,Y 391.25,Z 769.327,A -85,B 0,C 180,E1 21069.373,E2 21069.373} C_VEL
LIN {X 0,Y 401.63,Z 793.141,A -85,B 0,C 180,E1 21078.762,E2 21078.762} C_VEL
LIN {X 0,Y 412.153,Z 824.789,A -85,B 0,C 180,E1 21086.42,E2 21086.42} C_VEL
LIN {X 0,Y 414.926,Z 843.936,A -85,B 0,C 180,E1 21089.66,E2 21089.66} C_VEL
LIN {X 0,Y 388.207,Z 909.797,A -85,B 0,C 180,E1 21094.735,E2 21094.735} C_VEL
LIN {X 0,Y 366.289,Z 952.987,A -85,B 0,C 180,E1 21100.021,E2 21100.021} C_VEL
LIN {X 0,Y 347.302,Z 976.515,A -85,B 0,C 180,E1 21103.025,E2 21103.025} C_VEL
LIN {X 0,Y 321.15,Z 1019.625,A -85,B 0,C 180,E1 21113.828,E2 21113.828} C_VEL
LIN {X 0,Y 304.847,Z 1049.727,A -85,B 0,C 180,E1 21127.165,E2 21127.165} C_VEL
LIN {X 0,Y 299.617,Z 1064.519,A -85,B 0,C 180,E1 21139.797,E2 21139.797} C_VEL
LIN {X 0,Y 299.416,Z 1068.315,A -85,B 0,C 180,E1 21151.452,E2 21151.452} C_VEL
LIN {X 0,Y 300.685,Z 1061.824,A -85,B 0,C 180,E1 21164.606,E2 21164.606} C_VEL
LIN {X 0,Y 310.134,Z 1041.972,A -85,B 0,C 180,E1 21178.462,E2 21178.462} C_VEL
LIN {X 0,Y 332.851,Z 1006.63,A -85,B 0,C 180,E1 21191.346,E2 21191.346} C_VEL
LIN {X 0,Y 363.905,Z 958.068,A -85,B 0,C 180,E1 21201.283,E2 21201.283} C_VEL
LIN {X 0,Y 396.054,Z 899.513,A -85,B 0,C 180,E1 21208.16,E2 21208.16} C_VEL
LIN {X 0,Y 417.402,Z 850.016,A -85,B 0,C 180,E1 21211.802,E2 21211.802} C_VEL
LIN {X 0,Y 410.187,Z 818.775,A -85,B 0,C 180,E1 21219.395,E2 21219.395} C_VEL
LIN {X 0,Y 402.734,Z 797.174,A -85,B 0,C 180,E1 21228.013,E2 21228.013} C_VEL
LIN {X 0,Y 399.36,Z 787.457,A -85,B 0,C 180,E1 21236.708,E2 21236.708} C_VEL
LIN {X 0,Y 400.056,Z 790.496,A -85,B 0,C 180,E1 21244.328,E2 21244.328} C_VEL
LIN {X 0,Y 405.787,Z 806.032,A -85,B 0,C 180,E1 21253.495,E2 21253.495} C_VEL
LIN {X 0,Y 413.946,Z 835.148,A -85,B 0,C 180,E1 21262.285,E2 21262.285} C_VEL
LIN {X 0,Y 415.542,Z 852.417,A -85,B 0,C 180,E1 21265.681,E2 21265.681} C_VEL
LIN {X 0,Y 385.673,Z 916.99,A -85,B 0,C 180,E1 21271.046,E2 21271.046} C_VEL
LIN {X 0,Y 353.928,Z 970.93,A -85,B 0,C 180,E1 21278.726,E2 21278.726} C_VEL
LIN {X 0,Y 325.462,Z 1013.812,A -85,B 0,C 180,E1 21289.284,E2 21289.284} C_VEL
LIN {X 0,Y 307.077,Z 1042.984,A -85,B 0,C 180,E1 21302.021,E2 21302.021} C_VEL
LIN {X 0,Y 299.981,Z 1058.626,A -85,B 0,C 180,E1 21315.359,E2 21315.359} C_VEL
LIN {X 0,Y 299.247,Z 1062.342,A -85,B 0,C 180,E1 21328.547,E2 21328.547} C_VEL
LIN {X 0,Y 300.489,Z 1056.282,A -85,B 0,C 180,E1 21340.173,E2 21340.173} C_VEL
LIN {X 0,Y 308.873,Z 1036.914,A -85,B 0,C 180,E1 21353.893,E2 21353.893} C_VEL
LIN {X 0,Y 328.696,Z 1003.291,A -85,B 0,C 180,E1 21366.504,E2 21366.504} C_VEL
LIN {X 0,Y 357.354,Z 955.809,A -85,B 0,C 180,E1 21376.609,E2 21376.609} C_VEL
LIN {X 0,Y 387.961,Z 896.823,A -85,B 0,C 180,E1 21383.929,E2 21383.929} C_VEL
LIN {X 0,Y 409.067,Z 843.969,A -85,B 0,C 180,E1 21388.115,E2 21388.115} C_VEL
LIN {X 0,Y 400.089,Z 807.035,A -85,B 0,C 180,E1 21396.255,E2 21396.255} C_VEL
LIN {X 0,Y 390.67,Z 781.886,A -85,B 0,C 180,E1 21404.951,E2 21404.951} C_VEL
LIN {X 0,Y 385.556,Z 770.457,A -85,B 0,C 180,E1 21412.674,E2 21412.674} C_VEL
LIN {X 0,Y 384.844,Z 766.763,A -85,B 0,C 180,E1 21419.53,E2 21419.53} C_VEL
LIN {X 0,Y 388.654,Z 776.571,A -85,B 0,C 180,E1 21429.011,E2 21429.011} C_VEL
LIN {X 0,Y 398.048,Z 799.693,A -85,B 0,C 180,E1 21438.36,E2 21438.36} C_VEL
LIN {X 0,Y 407.896,Z 831.881,A -85,B 0,C 180,E1 21446.249,E2 21446.249} C_VEL
LIN {X 0,Y 409.314,Z 848.121,A -85,B 0,C 180,E1 21448.926,E2 21448.926} C_VEL
LIN {X 0,Y 381.313,Z 913.974,A -85,B 0,C 180,E1 21454.188,E2 21454.188} C_VEL
LIN {X 0,Y 350.881,Z 970.37,A -85,B 0,C 180,E1 21461.916,E2 21461.916} C_VEL
LIN {X 0,Y 347.302,Z 976.515,A -85,B 0,C 180,E1 21463.025,E2 21463.025} C_VEL
LIN {X 0,Y 328.573,Z 997.592,A -85,B 0,C 180,E1 21466.683,E2 21466.683} C_VEL
LIN {X 0,Y 305.711,Z 1034.328,A -85,B 0,C 180,E1 21478.613,E2 21478.613} C_VEL
LIN {X 0,Y 293.875,Z 1057.208,A -85,B 0,C 180,E1 21491.967,E2 21491.967} C_VEL
LIN {X 0,Y 291.229,Z 1066.188,A -85,B 0,C 180,E1 21502.521,E2 21502.521} C_VEL
LIN {X 0,Y 291.111,Z 1067.841,A -85,B 0,C 180,E1 21514.482,E2 21514.482} C_VEL
LIN {X 0,Y 293.805,Z 1058.853,A -85,B 0,C 180,E1 21527.885,E2 21527.885} C_VEL
LIN {X 0,Y 307.271,Z 1035.21,A -85,B 0,C 180,E1 21542.403,E2 21542.403} C_VEL
LIN {X 0,Y 333.415,Z 996.91,A -85,B 0,C 180,E1 21554.827,E2 21554.827} C_VEL
LIN {X 0,Y 365.703,Z 946.911,A -85,B 0,C 180,E1 21563.959,E2 21563.959} C_VEL
LIN {X 0,Y 397.995,Z 886.98,A -85,B 0,C 180,E1 21570.231,E2 21570.231} C_VEL
LIN {X 0,Y 412.011,Z 852.311,A -85,B 0,C 180,E1 21572.898,E2 21572.898} C_VEL
LIN {X 0,Y 405.069,Z 821.273,A -85,B 0,C 180,E1 21581.047,E2 21581.047} C_VEL
LIN {X 0,Y 398.634,Z 801.218,A -85,B 0,C 180,E1 21590.111,E2 21590.111} C_VEL
LIN {X 0,Y 396.801,Z 795.016,A -85,B 0,C 180,E1 21596.687,E2 21596.687} C_VEL
LIN {X 0,Y 397.3,Z 798.119,A -85,B 0,C 180,E1 21604.358,E2 21604.358} C_VEL
LIN {X 0,Y 402.685,Z 813.931,A -85,B 0,C 180,E1 21613.619,E2 21613.619} C_VEL
LIN {X 0,Y 409.789,Z 842.813,A -85,B 0,C 180,E1 21622.287,E2 21622.287} C_VEL
LIN {X 0,Y 410.567,Z 855.772,A -85,B 0,C 180,E1 21624.88,E2 21624.88} C_VEL
LIN {X 0,Y 379.734,Z 920.037,A -85,B 0,C 180,E1 21630.326,E2 21630.326} C_VEL
LIN {X 0,Y 346.457,Z 974.221,A -85,B 0,C 180,E1 21638.307,E2 21638.307} C_VEL
LIN {X 0,Y 317.707,Z 1015.727,A -85,B 0,C 180,E1 21648.982,E2 21648.982} C_VEL
LIN {X 0,Y 298.398,Z 1045.341,A -85,B 0,C 180,E1 21662.82,E2 21662.82} C_VEL
LIN {X 0,Y 291.706,Z 1059.604,A -85,B 0,C 180,E1 21676.471,E2 21676.471} C_VEL
LIN {X 0,Y 291.253,Z 1062.425,A -85,B 0,C 180,E1 21688.508,E2 21688.508} C_VEL
LIN {X 0,Y 292.56,Z 1056.399,A -85,B 0,C 180,E1 21700.451,E2 21700.451} C_VEL
LIN {X 0,Y 301.423,Z 1037.08,A -85,B 0,C 180,E1 21714.521,E2 21714.521} C_VEL
LIN {X 0,Y 322.012,Z 1003.712,A -85,B 0,C 180,E1 21727.322,E2 21727.322} C_VEL
LIN {X 0,Y 351.803,Z 956.109,A -85,B 0,C 180,E1 21737.574,E2 21737.574} C_VEL
LIN {X 0,Y 383.086,Z 897.593,A -85,B 0,C 180,E1 21744.867,E2 21744.867} C_VEL
LIN {X 0,Y 403.807,Z 848.323,A -85,B 0,C 180,E1 21748.731,E2 21748.731} C_VEL
LIN {X 0,Y 395.929,Z 812.568,A -85,B 0,C 180,E1 21756.889,E2 21756.889} C_VEL
LIN {X 0,Y 387.185,Z 787.955,A -85,B 0,C 180,E1 21765.843,E2 21765.843} C_VEL
LIN {X 0,Y 383.572,Z 778.487,A -85,B 0,C 180,E1 21772.064,E2 21772.064} C_VEL
LIN {X 0,Y 382.596,Z 774.595,A -85,B 0,C 180,E1 21779.598,E2 21779.598} C_VEL
LIN {X 0,Y 386.104,Z 784.405,A -85,B 0,C 180,E1 21789.072,E2 21789.072} C_VEL
LIN {X 0,Y 394.974,Z 808.018,A -85,B 0,C 180,E1 21798.508,E2 21798.508} C_VEL
LIN {X 0,Y 403.572,Z 839.819,A -85,B 0,C 180,E1 21806.288,E2 21806.288} C_VEL
LIN {X 0,Y 404.068,Z 851.135,A -85,B 0,C 180,E1 21808.126,E2 21808.126} C_VEL
LIN {X 0,Y 375.543,Z 915.969,A -85,B 0,C 180,E1 21813.396,E2 21813.396} C_VEL
LIN {X 0,Y 343.834,Z 972.675,A -85,B 0,C 180,E1 21821.349,E2 21821.349} C_VEL
LIN {X 0,Y 328.573,Z 997.592,A -85,B 0,C 180,E1 21826.683,E2 21826.683} C_VEL
LIN {X 0,Y 309.866,Z 1016.14,A -85,B 0,C 180,E1 21830.96,E2 21830.96} C_VEL
LIN {X 0,Y 290.769,Z 1047.318,A -85,B 0,C 180,E1 21844.517,E2 21844.517} C_VEL
LIN {X 0,Y 283.699,Z 1064.303,A -85,B 0,C 180,E1 21859.218,E2 21859.218} C_VEL
LIN {X 0,Y 283.413,Z 1068.167,A -85,B 0,C 180,E1 21871.534,E2 21871.534} C_VEL
LIN {X 0,Y 284.903,Z 1061.745,A -85,B 0,C 180,E1 21885.409,E2 21885.409} C_VEL
LIN {X 0,Y 295.644,Z 1041.929,A -85,B 0,C 180,E1 21900.007,E2 21900.007} C_VEL
LIN {X 0,Y 320.582,Z 1006.718,A -85,B 0,C 180,E1 21913.306,E2 21913.306} C_VEL
LIN {X 0,Y 354.056,Z 957.911,A -85,B 0,C 180,E1 21923.424,E2 21923.424} C_VEL
LIN {X 0,Y 387.734,Z 899.884,A -85,B 0,C 180,E1 21930.199,E2 21930.199} C_VEL
LIN {X 0,Y 407.121,Z 857.714,A -85,B 0,C 180,E1 21933.35,E2 21933.35} C_VEL
LIN {X 0,Y 401.39,Z 828.33,A -85,B 0,C 180,E1 21941.227,E2 21941.227} C_VEL
LIN {X 0,Y 395.694,Z 808.884,A -85,B 0,C 180,E1 21950.036,E2 21950.036} C_VEL
LIN {X 0,Y 393.906,Z 802.482,A -85,B 0,C 180,E1 21956.663,E2 21956.663} C_VEL
LIN {X 0,Y 394.373,Z 805.66,A -85,B 0,C 180,E1 21964.391,E2 21964.391} C_VEL
LIN {X 0,Y 398.941,Z 820.454,A -85,B 0,C 180,E1 21973.206,E2 21973.206} C_VEL
LIN {X 0,Y 405.048,Z 848.096,A -85,B 0,C 180,E1 21981.753,E2 21981.753} C_VEL
LIN {X 0,Y 405.68,Z 859.063,A -85,B 0,C 180,E1 21984.05,E2 21984.05} C_VEL
LIN {X 0,Y 373.831,Z 922.88,A -85,B 0,C 180,E1 21989.577,E2 21989.577} C_VEL
LIN {X 0,Y 339.893,Z 976.14,A -85,B 0,C 180,E1 21997.61,E2 21997.61} C_VEL
LIN {X 0,Y 309.229,Z 1018.66,A -85,B 0,C 180,E1 22009.03,E2 22009.03} C_VEL
LIN {X 0,Y 290.333,Z 1046.47,A -85,B 0,C 180,E1 22022.824,E2 22022.824} C_VEL
LIN {X 0,Y 283.767,Z 1059.656,A -85,B 0,C 180,E1 22036.085,E2 22036.085} C_VEL
LIN {X 0,Y 283.237,Z 1062.509,A -85,B 0,C 180,E1 22048.465,E2 22048.465} C_VEL
LIN {X 0,Y 284.647,Z 1056.516,A -85,B 0,C 180,E1 22060.745,E2 22060.745} C_VEL
LIN {X 0,Y 294.499,Z 1036.392,A -85,B 0,C 180,E1 22075.663,E2 22075.663} C_VEL
LIN {X 0,Y 317.057,Z 1001.57,A -85,B 0,C 180,E1 22088.883,E2 22088.883} C_VEL
LIN {X 0,Y 348.436,Z 952.941,A -85,B 0,C 180,E1 22099.127,E2 22099.127} C_VEL
LIN {X 0,Y 380.659,Z 893.722,A -85,B 0,C 180,E1 22106.253,E2 22106.253} C_VEL
LIN {X 0,Y 398.431,Z 851.428,A -85,B 0,C 180,E1 22109.613,E2 22109.613} C_VEL
LIN {X 0,Y 391.436,Z 817.379,A -85,B 0,C 180,E1 22117.736,E2 22117.736} C_VEL
LIN {X 0,Y 383.454,Z 792.333,A -85,B 0,C 180,E1 22127.451,E2 22127.451} C_VEL
LIN {X 0,Y 380.057,Z 782.707,A -85,B 0,C 180,E1 22136.591,E2 22136.591} C_VEL
LIN {X 0,Y 380.64,Z 785.039,A -85,B 0,C 180,E1 22143.454,E2 22143.454} C_VEL
LIN {X 0,Y 385.958,Z 799.13,A -85,B 0,C 180,E1 22152.516,E2 22152.516} C_VEL
LIN {X 0,Y 395.024,Z 827.22,A -85,B 0,C 180,E1 22161.73,E2 22161.73} C_VEL
LIN {X 0,Y 398.885,Z 854.153,A -85,B 0,C 180,E1 22167.301,E2 22167.301} C_VEL
LIN {X 0,Y 368.732,Z 920.109,A -85,B 0,C 180,E1 22172.809,E2 22172.809} C_VEL
LIN {X 0,Y 336.231,Z 975.901,A -85,B 0,C 180,E1 22180.922,E2 22180.922} C_VEL
LIN {X 0,Y 309.866,Z 1016.14,A -85,B 0,C 180,E1 22190.96,E2 22190.96} C_VEL
LIN {X 0,Y 292.804,Z 1032.011,A -85,B 0,C 180,E1 22196.061,E2 22196.061} C_VEL
LIN {X 0,Y 278.375,Z 1056.951,A -85,B 0,C 180,E1 22210.924,E2 22210.924} C_VEL
LIN {X 0,Y 275.246,Z 1065.989,A -85,B 0,C 180,E1 22222.084,E2 22222.084} C_VEL
LIN {X 0,Y 275.129,Z 1067.709,A -85,B 0,C 180,E1 22234.743,E2 22234.743} C_VEL
LIN {X 0,Y 278.323,Z 1058.614,A -85,B 0,C 180,E1 22249.082,E2 22249.082} C_VEL
LIN {X 0,Y 294.076,Z 1034.43,A -85,B 0,C 180,E1 22264.502,E2 22264.502} C_VEL
LIN {X 0,Y 322.84,Z 995.703,A -85,B 0,C 180,E1 22277.217,E2 22277.217} C_VEL
LIN {X 0,Y 357.515,Z 945.196,A -85,B 0,C 180,E1 22286.361,E2 22286.361} C_VEL
LIN {X 0,Y 391.801,Z 884.177,A -85,B 0,C 180,E1 22292.549,E2 22292.549} C_VEL
LIN {X 0,Y 402.041,Z 861.182,A -85,B 0,C 180,E1 22294.243,E2 22294.243} C_VEL
LIN {X 0,Y 397.001,Z 833.116,A -85,B 0,C 180,E1 22302.166,E2 22302.166} C_VEL
LIN {X 0,Y 392.172,Z 815.169,A -85,B 0,C 180,E1 22310.958,E2 22310.958} C_VEL
LIN {X 0,Y 390.797,Z 809.83,A -85,B 0,C 180,E1 22318.863,E2 22318.863} C_VEL
LIN {X 0,Y 392.579,Z 817.116,A -85,B 0,C 180,E1 22327.753,E2 22327.753} C_VEL
LIN {X 0,Y 397.517,Z 837.367,A -85,B 0,C 180,E1 22336.616,E2 22336.616} C_VEL
LIN {X 0,Y 401.172,Z 861.576,A -85,B 0,C 180,E1 22343.164,E2 22343.164} C_VEL
LIN {X 0,Y 368.478,Z 924.855,A -85,B 0,C 180,E1 22348.707,E2 22348.707} C_VEL
LIN {X 0,Y 333.905,Z 977.292,A -85,B 0,C 180,E1 22356.723,E2 22356.723} C_VEL
LIN {X 0,Y 302.481,Z 1019.178,A -85,B 0,C 180,E1 22368.188,E2 22368.188} C_VEL
LIN {X 0,Y 282.291,Z 1047.599,A -85,B 0,C 180,E1 22382.831,E2 22382.831} C_VEL
LIN {X 0,Y 275.836,Z 1059.707,A -85,B 0,C 180,E1 22395.676,E2 22395.676} C_VEL
LIN {X 0,Y 275.252,Z 1062.592,A -85,B 0,C 180,E1 22408.421,E2 22408.421} C_VEL
LIN {X 0,Y 276.726,Z 1056.633,A -85,B 0,C 180,E1 22421.057,E2 22421.057} C_VEL
LIN {X 0,Y 286.859,Z 1037.028,A -85,B 0,C 180,E1 22436.099,E2 22436.099} C_VEL
LIN {X 0,Y 309.929,Z 1002.989,A -85,B 0,C 180,E1 22449.498,E2 22449.498} C_VEL
LIN {X 0,Y 342.176,Z 954.811,A -85,B 0,C 180,E1 22459.904,E2 22459.904} C_VEL
LIN {X 0,Y 374.983,Z 896.582,A -85,B 0,C 180,E1 22467.044,E2 22467.044} C_VEL
LIN {X 0,Y 393.258,Z 855.632,A -85,B 0,C 180,E1 22470.297,E2 22470.297} C_VEL
LIN {X 0,Y 387.023,Z 822.016,A -85,B 0,C 180,E1 22478.641,E2 22478.641} C_VEL
LIN {X 0,Y 380.027,Z 798.364,A -85,B 0,C 180,E1 22488.389,E2 22488.389} C_VEL
LIN {X 0,Y 377.715,Z 789.208,A -85,B 0,C 180,E1 22498.874,E2 22498.874} C_VEL
LIN {X 0,Y 380.679,Z 799.985,A -85,B 0,C 180,E1 22509.202,E2 22509.202} C_VEL
LIN {X 0,Y 388.065,Z 823.574,A -85,B 0,C 180,E1 22518.553,E2 22518.553} C_VEL
LIN {X 0,Y 394.44,Z 855.176,A -85,B 0,C 180,E1 22526.291,E2 22526.291} C_VEL
LIN {X 0,Y 363.71,Z 920.952,A -85,B 0,C 180,E1 22531.845,E2 22531.845} C_VEL
LIN {X 0,Y 330.857,Z 975.651,A -85,B 0,C 180,E1 22539.837,E2 22539.837} C_VEL
LIN {X 0,Y 301.293,Z 1019.079,A -85,B 0,C 180,E1 22551.015,E2 22551.015} C_VEL
LIN {X 0,Y 292.804,Z 1032.011,A -85,B 0,C 180,E1 22556.061,E2 22556.061} C_VEL
LIN {X 0,Y 277.07,Z 1045.11,A -85,B 0,C 180,E1 22561.916,E2 22561.916} C_VEL
LIN {X 0,Y 268.116,Z 1062.858,A -85,B 0,C 180,E1 22576.925,E2 22576.925} C_VEL
LIN {X 0,Y 267.041,Z 1067.85,A -85,B 0,C 180,E1 22588.374,E2 22588.374} C_VEL
LIN {X 0,Y 267.858,Z 1064.995,A -85,B 0,C 180,E1 22601.429,E2 22601.429} C_VEL
LIN {X 0,Y 276.158,Z 1049.592,A -85,B 0,C 180,E1 22616.938,E2 22616.938} C_VEL
LIN {X 0,Y 298.609,Z 1019.747,A -85,B 0,C 180,E1 22631.314,E2 22631.314} C_VEL
LIN {X 0,Y 332.177,Z 975.903,A -85,B 0,C 180,E1 22642.583,E2 22642.583} C_VEL
LIN {X 0,Y 368.149,Z 921.035,A -85,B 0,C 180,E1 22650.365,E2 22650.365} C_VEL
LIN {X 0,Y 396.935,Z 864.603,A -85,B 0,C 180,E1 22655.19,E2 22655.19} C_VEL
LIN {X 0,Y 392.598,Z 837.931,A -85,B 0,C 180,E1 22663.12,E2 22663.12} C_VEL
LIN {X 0,Y 388.465,Z 821.246,A -85,B 0,C 180,E1 22672.116,E2 22672.116} C_VEL
LIN {X 0,Y 387.665,Z 817.191,A -85,B 0,C 180,E1 22678.854,E2 22678.854} C_VEL
LIN {X 0,Y 389.265,Z 824.676,A -85,B 0,C 180,E1 22687.819,E2 22687.819} C_VEL
LIN {X 0,Y 393.671,Z 845.354,A -85,B 0,C 180,E1 22696.783,E2 22696.783} C_VEL
LIN {X 0,Y 395.92,Z 865.733,A -85,B 0,C 180,E1 22702.376,E2 22702.376} C_VEL
LIN {X 0,Y 361.961,Z 928.916,A -85,B 0,C 180,E1 22708.066,E2 22708.066} C_VEL
LIN {X 0,Y 326.263,Z 980.92,A -85,B 0,C 180,E1 22716.335,E2 22716.335} C_VEL
LIN {X 0,Y 293.926,Z 1022.168,A -85,B 0,C 180,E1 22728.247,E2 22728.247} C_VEL
LIN {X 0,Y 274.864,Z 1047.605,A -85,B 0,C 180,E1 22742.034,E2 22742.034} C_VEL
LIN {X 0,Y 267.919,Z 1059.759,A -85,B 0,C 180,E1 22755.243,E2 22755.243} C_VEL
LIN {X 0,Y 267.234,Z 1062.675,A -85,B 0,C 180,E1 22768.373,E2 22768.373} C_VEL
LIN {X 0,Y 268.823,Z 1056.749,A -85,B 0,C 180,E1 22781.386,E2 22781.386} C_VEL
LIN {X 0,Y 279.296,Z 1037.571,A -85,B 0,C 180,E1 22796.612,E2 22796.612} C_VEL
LIN {X 0,Y 302.854,Z 1004.382,A -85,B 0,C 180,E1 22810.139,E2 22810.139} C_VEL
LIN {X 0,Y 335.319,Z 957.746,A -85,B 0,C 180,E1 22820.534,E2 22820.534} C_VEL
LIN {X 0,Y 368.818,Z 900.474,A -85,B 0,C 180,E1 22827.771,E2 22827.771} C_VEL
LIN {X 0,Y 387.914,Z 858.183,A -85,B 0,C 180,E1 22831.367,E2 22831.367} C_VEL
LIN {X 0,Y 382.525,Z 826.347,A -85,B 0,C 180,E1 22839.711,E2 22839.711} C_VEL
LIN {X 0,Y 376.442,Z 804.238,A -85,B 0,C 180,E1 22849.572,E2 22849.572} C_VEL
LIN {X 0,Y 375.06,Z 796.774,A -85,B 0,C 180,E1 22858.866,E2 22858.866} C_VEL
LIN {X 0,Y 377.69,Z 807.763,A -85,B 0,C 180,E1 22869.275,E2 22869.275} C_VEL
LIN {X 0,Y 384.326,Z 830.88,A -85,B 0,C 180,E1 22878.443,E2 22878.443} C_VEL
LIN {X 0,Y 389.105,Z 859.519,A -85,B 0,C 180,E1 22885.562,E2 22885.562} C_VEL
LIN {X 0,Y 357.511,Z 924.125,A -85,B 0,C 180,E1 22891.101,E2 22891.101} C_VEL
LIN {X 0,Y 323.2,Z 978.794,A -85,B 0,C 180,E1 22899.382,E2 22899.382} C_VEL
LIN {X 0,Y 293.061,Z 1021.342,A -85,B 0,C 180,E1 22910.891,E2 22910.891} C_VEL
LIN {X 0,Y 277.07,Z 1045.11,A -85,B 0,C 180,E1 22921.916,E2 22921.916} C_VEL
LIN {X 0,Y 263.715,Z 1055.301,A -85,B 0,C 180,E1 22928.562,E2 22928.562} C_VEL
LIN {X 0,Y 259.277,Z 1065.79,A -85,B 0,C 180,E1 22941.593,E2 22941.593} C_VEL
LIN {X 0,Y 259.131,Z 1067.575,A -85,B 0,C 180,E1 22955.037,E2 22955.037} C_VEL
LIN {X 0,Y 262.893,Z 1058.533,A -85,B 0,C 180,E1 22970.249,E2 22970.249} C_VEL
LIN {X 0,Y 280.67,Z 1034.332,A -85,B 0,C 180,E1 22986.464,E2 22986.464} C_VEL
LIN {X 0,Y 311.812,Z 995.821,A -85,B 0,C 180,E1 22999.454,E2 22999.454} C_VEL
LIN {X 0,Y 349.285,Z 944.577,A -85,B 0,C 180,E1 23008.717,E2 23008.717} C_VEL
LIN {X 0,Y 384.684,Z 884.396,A -85,B 0,C 180,E1 23014.716,E2 23014.716} C_VEL
LIN {X 0,Y 391.87,Z 868.667,A -85,B 0,C 180,E1 23015.977,E2 23015.977} C_VEL
LIN {X 0,Y 388.188,Z 842.498,A -85,B 0,C 180,E1 23024.236,E2 23024.236} C_VEL
LIN {X 0,Y 384.953,Z 827.414,A -85,B 0,C 180,E1 23033.182,E2 23033.182} C_VEL
LIN {X 0,Y 384.622,Z 824.827,A -85,B 0,C 180,E1 23041.106,E2 23041.106} C_VEL
LIN {X 0,Y 386.825,Z 837.155,A -85,B 0,C 180,E1 23050.717,E2 23050.717} C_VEL
LIN {X 0,Y 390.486,Z 860.872,A -85,B 0,C 180,E1 23059.267,E2 23059.267} C_VEL
LIN {X 0,Y 389.945,Z 871.557,A -85,B 0,C 180,E1 23061.675,E2 23061.675} C_VEL
LIN {X 0,Y 354.804,Z 934.038,A -85,B 0,C 180,E1 23067.52,E2 23067.52} C_VEL
LIN {X 0,Y 317.334,Z 985.977,A -85,B 0,C 180,E1 23076.257,E2 23076.257} C_VEL
LIN {X 0,Y 285.265,Z 1024.982,A -85,B 0,C 180,E1 23088.357,E2 23088.357} C_VEL
LIN {X 0,Y 265.925,Z 1049.884,A -85,B 0,C 180,E1 23103.11,E2 23103.11} C_VEL
LIN {X 0,Y 259.291,Z 1061.448,A -85,B 0,C 180,E1 23118.188,E2 23118.188} C_VEL
LIN {X 0,Y 259.287,Z 1062.117,A -85,B 0,C 180,E1 23131.675,E2 23131.675} C_VEL
LIN {X 0,Y 262.949,Z 1052.345,A -85,B 0,C 180,E1 23146.758,E2 23146.758} C_VEL
LIN {X 0,Y 278.625,Z 1028.623,A -85,B 0,C 180,E1 23162.103,E2 23162.103} C_VEL
LIN {X 0,Y 307.645,Z 989.853,A -85,B 0,C 180,E1 23175.162,E2 23175.162} C_VEL
LIN {X 0,Y 342.41,Z 939.215,A -85,B 0,C 180,E1 23184.464,E2 23184.464} C_VEL
LIN {X 0,Y 375.853,Z 878.786,A -85,B 0,C 180,E1 23190.714,E2 23190.714} C_VEL
LIN {X 0,Y 382.724,Z 861.747,A -85,B 0,C 180,E1 23192.24,E2 23192.24} C_VEL
LIN {X 0,Y 378.141,Z 831.144,A -85,B 0,C 180,E1 23200.627,E2 23200.627} C_VEL
LIN {X 0,Y 373.098,Z 810.161,A -85,B 0,C 180,E1 23210.661,E2 23210.661} C_VEL
LIN {X 0,Y 372.142,Z 804.271,A -85,B 0,C 180,E1 23218.857,E2 23218.857} C_VEL
LIN {X 0,Y 374.603,Z 815.449,A -85,B 0,C 180,E1 23229.352,E2 23229.352} C_VEL
LIN {X 0,Y 380.626,Z 839.593,A -85,B 0,C 180,E1 23238.815,E2 23238.815} C_VEL
LIN {X 0,Y 383.327,Z 864.582,A -85,B 0,C 180,E1 23244.811,E2 23244.811} C_VEL
LIN {X 0,Y 350.727,Z 928.156,A -85,B 0,C 180,E1 23250.469,E2 23250.469} C_VEL
LIN {X 0,Y 315.432,Z 982.13,A -85,B 0,C 180,E1 23258.971,E2 23258.971} C_VEL
LIN {X 0,Y 284.01,Z 1024.814,A -85,B 0,C 180,E1 23271.227,E2 23271.227} C_VEL
LIN {X 0,Y 265.473,Z 1052.055,A -85,B 0,C 180,E1 23285.881,E2 23285.881} C_VEL
LIN {X 0,Y 263.715,Z 1055.301,A -85,B 0,C 180,E1 23288.562,E2 23288.562} C_VEL
LIN {X 0,Y 252.355,Z 1062.493,A -85,B 0,C 180,E1 23295.882,E2 23295.882} C_VEL
LIN {X 0,Y 251.032,Z 1067.686,A -85,B 0,C 180,E1 23308.27,E2 23308.27} C_VEL
LIN {X 0,Y 251.971,Z 1064.88,A -85,B 0,C 180,E1 23322.161,E2 23322.161} C_VEL
LIN {X 0,Y 261.462,Z 1049.549,A -85,B 0,C 180,E1 23338.587,E2 23338.587} C_VEL
LIN {X 0,Y 286.264,Z 1019.791,A -85,B 0,C 180,E1 23353.524,E2 23353.524} C_VEL
LIN {X 0,Y 322.06,Z 976.494,A -85,B 0,C 180,E1 23364.837,E2 23364.837} C_VEL
LIN {X 0,Y 360.181,Z 921.67,A -85,B 0,C 180,E1 23372.588,E2 23372.588} C_VEL
LIN {X 0,Y 386.839,Z 872.998,A -85,B 0,C 180,E1 23376.736,E2 23376.736} C_VEL
LIN {X 0,Y 383.956,Z 847.812,A -85,B 0,C 180,E1 23385.086,E2 23385.086} C_VEL
LIN {X 0,Y 381.429,Z 833.426,A -85,B 0,C 180,E1 23394.266,E2 23394.266} C_VEL
LIN {X 0,Y 381.232,Z 832.109,A -85,B 0,C 180,E1 23401.116,E2 23401.116} C_VEL
LIN {X 0,Y 383.242,Z 845.234,A -85,B 0,C 180,E1 23411.091,E2 23411.091} C_VEL
LIN {X 0,Y 385.909,Z 870.231,A -85,B 0,C 180,E1 23419.881,E2 23419.881} C_VEL
LIN {X 0,Y 384.396,Z 876.639,A -85,B 0,C 180,E1 23420.911,E2 23420.911} C_VEL
LIN {X 0,Y 348.312,Z 937.814,A -85,B 0,C 180,E1 23426.811,E2 23426.811} C_VEL
LIN {X 0,Y 310.194,Z 988.557,A -85,B 0,C 180,E1 23435.636,E2 23435.636} C_VEL
LIN {X 0,Y 277.497,Z 1026.698,A -85,B 0,C 180,E1 23447.977,E2 23447.977} C_VEL
LIN {X 0,Y 257.327,Z 1051.563,A -85,B 0,C 180,E1 23463.769,E2 23463.769} C_VEL
LIN {X 0,Y 251.339,Z 1061.511,A -85,B 0,C 180,E1 23477.808,E2 23477.808} C_VEL
LIN {X 0,Y 251.286,Z 1062.211,A -85,B 0,C 180,E1 23491.728,E2 23491.728} C_VEL
LIN {X 0,Y 255.15,Z 1052.575,A -85,B 0,C 180,E1 23507.201,E2 23507.201} C_VEL
LIN {X 0,Y 271.75,Z 1028.811,A -85,B 0,C 180,E1 23523.017,E2 23523.017} C_VEL
LIN {X 0,Y 301.857,Z 990.216,A -85,B 0,C 180,E1 23536.231,E2 23536.231} C_VEL
LIN {X 0,Y 337.763,Z 939.528,A -85,B 0,C 180,E1 23545.583,E2 23545.583} C_VEL
LIN {X 0,Y 371.466,Z 880.224,A -85,B 0,C 180,E1 23551.714,E2 23551.714} C_VEL
LIN {X 0,Y 377.579,Z 866.416,A -85,B 0,C 180,E1 23552.859,E2 23552.859} C_VEL
LIN {X 0,Y 373.91,Z 836.914,A -85,B 0,C 180,E1 23561.23,E2 23561.23} C_VEL
LIN {X 0,Y 369.867,Z 817.749,A -85,B 0,C 180,E1 23570.578,E2 23570.578} C_VEL
LIN {X 0,Y 369.231,Z 811.747,A -85,B 0,C 180,E1 23578.848,E2 23578.848} C_VEL
LIN {X 0,Y 370.744,Z 821.101,A -85,B 0,C 180,E1 23588.264,E2 23588.264} C_VEL
LIN {X 0,Y 375.842,Z 843.382,A -85,B 0,C 180,E1 23597.657,E2 23597.657} C_VEL
LIN {X 0,Y 378.762,Z 866.716,A -85,B 0,C 180,E1 23603.859,E2 23603.859} C_VEL
LIN {X 0,Y 345.572,Z 929.538,A -85,B 0,C 180,E1 23609.493,E2 23609.493} C_VEL
LIN {X 0,Y 308.957,Z 983.66,A -85,B 0,C 180,E1 23618.148,E2 23618.148} C_VEL
LIN {X 0,Y 277.547,Z 1024.63,A -85,B 0,C 180,E1 23630.147,E2 23630.147} C_VEL
LIN {X 0,Y 257.875,Z 1052.035,A -85,B 0,C 180,E1 23645.218,E2 23645.218} C_VEL
LIN {X 0,Y 252.355,Z 1062.493,A -85,B 0,C 180,E1 23655.882,E2 23655.882} C_VEL
LIN {X 0,Y 243.006,Z 1066.569,A -85,B 0,C 180,E1 23663.787,E2 23663.787} C_VEL
LIN {X 0,Y 243.119,Z 1067.436,A -85,B 0,C 180,E1 23675.369,E2 23675.369} C_VEL
LIN {X 0,Y 247.588,Z 1058.454,A -85,B 0,C 180,E1 23691.561,E2 23691.561} C_VEL
LIN {X 0,Y 267.514,Z 1034.332,A -85,B 0,C 180,E1 23708.576,E2 23708.576} C_VEL
LIN {X 0,Y 301.233,Z 996.044,A -85,B 0,C 180,E1 23721.822,E2 23721.822} C_VEL
LIN {X 0,Y 340.434,Z 945.739,A -85,B 0,C 180,E1 23730.948,E2 23730.948} C_VEL
LIN {X 0,Y 377.885,Z 885.146,A -85,B 0,C 180,E1 23736.911,E2 23736.911} C_VEL
LIN {X 0,Y 381.819,Z 876.353,A -85,B 0,C 180,E1 23737.786,E2 23737.786} C_VEL
LIN {X 0,Y 379.53,Z 852.81,A -85,B 0,C 180,E1 23746.09,E2 23746.09} C_VEL
LIN {X 0,Y 377.815,Z 840.725,A -85,B 0,C 180,E1 23754.211,E2 23754.211} C_VEL
LIN {X 0,Y 377.648,Z 839.311,A -85,B 0,C 180,E1 23761.126,E2 23761.126} C_VEL
LIN {X 0,Y 379.146,Z 852.189,A -85,B 0,C 180,E1 23770.989,E2 23770.989} C_VEL
LIN {X 0,Y 381.103,Z 876.996,A -85,B 0,C 180,E1 23779.761,E2 23779.761} C_VEL
LIN {X 0,Y 344.643,Z 937.657,A -85,B 0,C 180,E1 23785.578,E2 23785.578} C_VEL
LIN {X 0,Y 305.39,Z 988.471,A -85,B 0,C 180,E1 23794.358,E2 23794.358} C_VEL
LIN {X 0,Y 271.192,Z 1026.781,A -85,B 0,C 180,E1 23806.836,E2 23806.836} C_VEL
LIN {X 0,Y 249.871,Z 1051.582,A -85,B 0,C 180,E1 23822.924,E2 23822.924} C_VEL
LIN {X 0,Y 243.384,Z 1061.574,A -85,B 0,C 180,E1 23837.403,E2 23837.403} C_VEL
LIN {X 0,Y 243.303,Z 1062.305,A -85,B 0,C 180,E1 23851.785,E2 23851.785} C_VEL
LIN {X 0,Y 247.154,Z 1053.154,A -85,B 0,C 180,E1 23867.26,E2 23867.26} C_VEL
LIN {X 0,Y 264.658,Z 1029.372,A -85,B 0,C 180,E1 23883.805,E2 23883.805} C_VEL
LIN {X 0,Y 296.27,Z 990.458,A -85,B 0,C 180,E1 23897.371,E2 23897.371} C_VEL
LIN {X 0,Y 333.222,Z 939.842,A -85,B 0,C 180,E1 23906.74,E2 23906.74} C_VEL
LIN {X 0,Y 367.728,Z 880.635,A -85,B 0,C 180,E1 23912.816,E2 23912.816} C_VEL
LIN {X 0,Y 372.418,Z 870.056,A -85,B 0,C 180,E1 23913.751,E2 23913.751} C_VEL
LIN {X 0,Y 369.631,Z 841.979,A -85,B 0,C 180,E1 23922.09,E2 23922.09} C_VEL
LIN {X 0,Y 366.264,Z 823.849,A -85,B 0,C 180,E1 23931.686,E2 23931.686} C_VEL
LIN {X 0,Y 365.999,Z 819.114,A -85,B 0,C 180,E1 23938.838,E2 23938.838} C_VEL
LIN {X 0,Y 367.684,Z 829.644,A -85,B 0,C 180,E1 23948.931,E2 23948.931} C_VEL
LIN {X 0,Y 371.96,Z 852.394,A -85,B 0,C 180,E1 23958.174,E2 23958.174} C_VEL
LIN {X 0,Y 373.31,Z 870.932,A -85,B 0,C 180,E1 23963.024,E2 23963.024} C_VEL
LIN {X 0,Y 338.979,Z 933.347,A -85,B 0,C 180,E1 23968.773,E2 23968.773} C_VEL
LIN {X 0,Y 301.987,Z 985.95,A -85,B 0,C 180,E1 23977.454,E2 23977.454} C_VEL
LIN {X 0,Y 269.812,Z 1026.242,A -85,B 0,C 180,E1 23989.736,E2 23989.736} C_VEL
LIN {X 0,Y 249.581,Z 1053.217,A -85,B 0,C 180,E1 24005.512,E2 24005.512} C_VEL
LIN {X 0,Y 243.316,Z 1065.589,A -85,B 0,C 180,E1 24021.037,E2 24021.037} C_VEL
LIN {X 0,Y 243.006,Z 1066.569,A -85,B 0,C 180,E1 24023.787,E2 24023.787} C_VEL
LIN {X 0,Y 235.289,Z 1067.699,A -85,B 0,C 180,E1 24032.114,E2 24032.114} C_VEL
LIN {X 0,Y 237.929,Z 1061.431,A -85,B 0,C 180,E1 24048.583,E2 24048.583} C_VEL
LIN {X 0,Y 254.013,Z 1041.712,A -85,B 0,C 180,E1 24065.715,E2 24065.715} C_VEL
LIN {X 0,Y 286.391,Z 1006.997,A -85,B 0,C 180,E1 24080.154,E2 24080.154} C_VEL
LIN {X 0,Y 327.023,Z 958.612,A -85,B 0,C 180,E1 24090.371,E2 24090.371} C_VEL
LIN {X 0,Y 366.402,Z 900.305,A -85,B 0,C 180,E1 24096.889,E2 24096.889} C_VEL
LIN {X 0,Y 376.882,Z 881.117,A -85,B 0,C 180,E1 24098.45,E2 24098.45} C_VEL
LIN {X 0,Y 375.172,Z 857.897,A -85,B 0,C 180,E1 24107.118,E2 24107.118} C_VEL
LIN {X 0,Y 374.111,Z 846.323,A -85,B 0,C 180,E1 24116.486,E2 24116.486} C_VEL
LIN {X 0,Y 373.895,Z 849.498,A -85,B 0,C 180,E1 24124.481,E2 24124.481} C_VEL
LIN {X 0,Y 375.48,Z 864.895,A -85,B 0,C 180,E1 24133.414,E2 24133.414} C_VEL
LIN {X 0,Y 375.394,Z 882.444,A -85,B 0,C 180,E1 24139.056,E2 24139.056} C_VEL
LIN {X 0,Y 337.22,Z 942.856,A -85,B 0,C 180,E1 24145.001,E2 24145.001} C_VEL
LIN {X 0,Y 296.775,Z 992.891,A -85,B 0,C 180,E1 24154.112,E2 24154.112} C_VEL
LIN {X 0,Y 261.519,Z 1030.576,A -85,B 0,C 180,E1 24167.396,E2 24167.396} C_VEL
LIN {X 0,Y 241.07,Z 1053.406,A -85,B 0,C 180,E1 24183.875,E2 24183.875} C_VEL
LIN {X 0,Y 234.952,Z 1062.654,A -85,B 0,C 180,E1 24200.714,E2 24200.714} C_VEL
LIN {X 0,Y 235.307,Z 1062.232,A -85,B 0,C 180,E1 24212.448,E2 24212.448} C_VEL
LIN {X 0,Y 240.152,Z 1052.107,A -85,B 0,C 180,E1 24229.061,E2 24229.061} C_VEL
LIN {X 0,Y 259.604,Z 1027.571,A -85,B 0,C 180,E1 24245.74,E2 24245.74} C_VEL
LIN {X 0,Y 293.08,Z 987.924,A -85,B 0,C 180,E1 24259.241,E2 24259.241} C_VEL
LIN {X 0,Y 331.496,Z 936.353,A -85,B 0,C 180,E1 24268.428,E2 24268.428} C_VEL
LIN {X 0,Y 367.345,Z 873.797,A -85,B 0,C 180,E1 24274.645,E2 24274.645} C_VEL
LIN {X 0,Y 365.214,Z 846.779,A -85,B 0,C 180,E1 24283.114,E2 24283.114} C_VEL
LIN {X 0,Y 362.866,Z 831.299,A -85,B 0,C 180,E1 24291.608,E2 24291.608} C_VEL
LIN {X 0,Y 362.747,Z 826.465,A -85,B 0,C 180,E1 24298.827,E2 24298.827} C_VEL
LIN {X 0,Y 364.036,Z 837.095,A -85,B 0,C 180,E1 24309.021,E2 24309.021} C_VEL
LIN {X 0,Y 367.579,Z 859.39,A -85,B 0,C 180,E1 24318.067,E2 24318.067} C_VEL
LIN {X 0,Y 367.515,Z 876.054,A -85,B 0,C 180,E1 24322.23,E2 24322.23} C_VEL
LIN {X 0,Y 331.712,Z 938.289,A -85,B 0,C 180,E1 24328.168,E2 24328.168} C_VEL
LIN {X 0,Y 293.116,Z 990.545,A -85,B 0,C 180,E1 24337.307,E2 24337.307} C_VEL
LIN {X 0,Y 260.456,Z 1029.6,A -85,B 0,C 180,E1 24350.177,E2 24350.177} C_VEL
LIN {X 0,Y 241.225,Z 1054.392,A -85,B 0,C 180,E1 24365.926,E2 24365.926} C_VEL
LIN {X 0,Y 235.355,Z 1065.489,A -85,B 0,C 180,E1 24380.731,E2 24380.731} C_VEL
LIN {X 0,Y 235.289,Z 1067.699,A -85,B 0,C 180,E1 24392.114,E2 24392.114} C_VEL
LIN {X 0,Y 227.544,Z 1065.83,A -85,B 0,C 180,E1 24400.682,E2 24400.682} C_VEL
LIN {X 0,Y 237.066,Z 1052.864,A -85,B 0,C 180,E1 24418.67,E2 24418.67} C_VEL
LIN {X 0,Y 263.999,Z 1024.829,A -85,B 0,C 180,E1 24435.244,E2 24435.244} C_VEL
LIN {X 0,Y 303.541,Z 982.396,A -85,B 0,C 180,E1 24447.463,E2 24447.463} C_VEL
LIN {X 0,Y 344.926,Z 928.984,A -85,B 0,C 180,E1 24455.437,E2 24455.437} C_VEL
LIN {X 0,Y 371.875,Z 885.031,A -85,B 0,C 180,E1 24459.362,E2 24459.362} C_VEL
LIN {X 0,Y 370.896,Z 863.032,A -85,B 0,C 180,E1 24468.167,E2 24468.167} C_VEL
LIN {X 0,Y 370.209,Z 853.367,A -85,B 0,C 180,E1 24476.449,E2 24476.449} C_VEL
LIN {X 0,Y 369.973,Z 856.584,A -85,B 0,C 180,E1 24484.528,E2 24484.528} C_VEL
LIN {X 0,Y 371.006,Z 871.971,A -85,B 0,C 180,E1 24493.432,E2 24493.432} C_VEL
LIN {X 0,Y 370.7,Z 885.928,A -85,B 0,C 180,E1 24498.129,E2 24498.129} C_VEL
LIN {X 0,Y 331.735,Z 945.482,A -85,B 0,C 180,E1 24504.066,E2 24504.066} C_VEL
LIN {X 0,Y 290.284,Z 994.888,A -85,B 0,C 180,E1 24513.26,E2 24513.26} C_VEL
LIN {X 0,Y 254.265,Z 1031.632,A -85,B 0,C 180,E1 24526.696,E2 24526.696} C_VEL
LIN {X 0,Y 233.629,Z 1053.437,A -85,B 0,C 180,E1 24542.976,E2 24542.976} C_VEL
LIN {X 0,Y 226.958,Z 1062.717,A -85,B 0,C 180,E1 24560.384,E2 24560.384} C_VEL
LIN {X 0,Y 227.341,Z 1062.492,A -85,B 0,C 180,E1 24571.91,E2 24571.91} C_VEL
LIN {X 0,Y 231.645,Z 1053.521,A -85,B 0,C 180,E1 24588.312,E2 24588.312} C_VEL
LIN {X 0,Y 251.53,Z 1029.473,A -85,B 0,C 180,E1 24606,E2 24606} C_VEL
LIN {X 0,Y 285.456,Z 990.943,A -85,B 0,C 180,E1 24619.785,E2 24619.785} C_VEL
LIN {X 0,Y 324.979,Z 939.936,A -85,B 0,C 180,E1 24629.207,E2 24629.207} C_VEL
LIN {X 0,Y 361.963,Z 879.047,A -85,B 0,C 180,E1 24635.269,E2 24635.269} C_VEL
LIN {X 0,Y 361.083,Z 854.103,A -85,B 0,C 180,E1 24643.066,E2 24643.066} C_VEL
LIN {X 0,Y 359.242,Z 838.659,A -85,B 0,C 180,E1 24651.523,E2 24651.523} C_VEL
LIN {X 0,Y 359.287,Z 833.726,A -85,B 0,C 180,E1 24658.816,E2 24658.816} C_VEL
LIN {X 0,Y 360.369,Z 844.557,A -85,B 0,C 180,E1 24669.114,E2 24669.114} C_VEL
LIN {X 0,Y 363.248,Z 868.294,A -85,B 0,C 180,E1 24678.606,E2 24678.606} C_VEL
LIN {X 0,Y 362.345,Z 879.963,A -85,B 0,C 180,E1 24681.331,E2 24681.331} C_VEL
LIN {X 0,Y 324.754,Z 942.427,A -85,B 0,C 180,E1 24687.479,E2 24687.479} C_VEL
LIN {X 0,Y 284.813,Z 994.36,A -85,B 0,C 180,E1 24697.001,E2 24697.001} C_VEL
LIN {X 0,Y 251.124,Z 1032.954,A -85,B 0,C 180,E1 24710.652,E2 24710.652} C_VEL
LIN {X 0,Y 232.321,Z 1056.331,A -85,B 0,C 180,E1 24727.105,E2 24727.105} C_VEL
LIN {X 0,Y 227.023,Z 1066.687,A -85,B 0,C 180,E1 24744.251,E2 24744.251} C_VEL
LIN {X 0,Y 227.099,Z 1067.293,A -85,B 0,C 180,E1 24755.749,E2 24755.749} C_VEL
LIN {X 0,Y 227.544,Z 1065.83,A -85,B 0,C 180,E1 24760.682,E2 24760.682} C_VEL
LIN {X 0,Y 222.317,Z 1061.534,A -85,B 0,C 180,E1 24769.603,E2 24769.603} C_VEL
LIN {X 0,Y 240.56,Z 1041.902,A -85,B 0,C 180,E1 24787.875,E2 24787.875} C_VEL
LIN {X 0,Y 276.102,Z 1007.095,A -85,B 0,C 180,E1 24802.786,E2 24802.786} C_VEL
LIN {X 0,Y 318.788,Z 959.375,A -85,B 0,C 180,E1 24812.855,E2 24812.855} C_VEL
LIN {X 0,Y 360.159,Z 900.977,A -85,B 0,C 180,E1 24819.243,E2 24819.243} C_VEL
LIN {X 0,Y 366.902,Z 888.727,A -85,B 0,C 180,E1 24820.401,E2 24820.401} C_VEL
LIN {X 0,Y 366.461,Z 868.157,A -85,B 0,C 180,E1 24829.232,E2 24829.232} C_VEL
LIN {X 0,Y 366.295,Z 860.428,A -85,B 0,C 180,E1 24836.411,E2 24836.411} C_VEL
LIN {X 0,Y 365.987,Z 862.6,A -85,B 0,C 180,E1 24843.541,E2 24843.541} C_VEL
LIN {X 0,Y 366.44,Z 876.849,A -85,B 0,C 180,E1 24852.533,E2 24852.533} C_VEL
LIN {X 0,Y 364.99,Z 891.414,A -85,B 0,C 180,E1 24857.329,E2 24857.329} C_VEL
LIN {X 0,Y 324.682,Z 950.138,A -85,B 0,C 180,E1 24863.381,E2 24863.381} C_VEL
LIN {X 0,Y 282.088,Z 998.502,A -85,B 0,C 180,E1 24872.854,E2 24872.854} C_VEL
LIN {X 0,Y 244.98,Z 1034.695,A -85,B 0,C 180,E1 24887.085,E2 24887.085} C_VEL
LIN {X 0,Y 224.788,Z 1055.029,A -85,B 0,C 180,E1 24903.992,E2 24903.992} C_VEL
LIN {X 0,Y 218.968,Z 1062.78,A -85,B 0,C 180,E1 24920.029,E2 24920.029} C_VEL
LIN {X 0,Y 219.35,Z 1062.585,A -85,B 0,C 180,E1 24931.98,E2 24931.98} C_VEL
LIN {X 0,Y 223.949,Z 1053.648,A -85,B 0,C 180,E1 24948.965,E2 24948.965} C_VEL
LIN {X 0,Y 244.963,Z 1029.66,A -85,B 0,C 180,E1 24967.124,E2 24967.124} C_VEL
LIN {X 0,Y 280.245,Z 991.184,A -85,B 0,C 180,E1 24981.062,E2 24981.062} C_VEL
LIN {X 0,Y 320.79,Z 940.427,A -85,B 0,C 180,E1 24990.42,E2 24990.42} C_VEL
LIN {X 0,Y 357.234,Z 881.227,A -85,B 0,C 180,E1 24996.494,E2 24996.494} C_VEL
LIN {X 0,Y 356.455,Z 857.099,A -85,B 0,C 180,E1 25004.912,E2 25004.912} C_VEL
LIN {X 0,Y 355.302,Z 844.481,A -85,B 0,C 180,E1 25013.129,E2 25013.129} C_VEL
LIN {X 0,Y 355.713,Z 840.909,A -85,B 0,C 180,E1 25018.804,E2 25018.804} C_VEL
LIN {X 0,Y 356.43,Z 851.939,A -85,B 0,C 180,E1 25029.215,E2 25029.215} C_VEL
LIN {X 0,Y 358.494,Z 875.296,A -85,B 0,C 180,E1 25038.542,E2 25038.542} C_VEL
LIN {X 0,Y 357.513,Z 883.116,A -85,B 0,C 180,E1 25040.375,E2 25040.375} C_VEL
LIN {X 0,Y 319.62,Z 944.082,A -85,B 0,C 180,E1 25046.427,E2 25046.427} C_VEL
LIN {X 0,Y 278.725,Z 995.48,A -85,B 0,C 180,E1 25055.976,E2 25055.976} C_VEL
LIN {X 0,Y 243.36,Z 1034.28,A -85,B 0,C 180,E1 25070.184,E2 25070.184} C_VEL
LIN {X 0,Y 223.573,Z 1057.824,A -85,B 0,C 180,E1 25088.098,E2 25088.098} C_VEL
LIN {X 0,Y 219.019,Z 1066.595,A -85,B 0,C 180,E1 25104.04,E2 25104.04} C_VEL
LIN {X 0,Y 219.118,Z 1067.219,A -85,B 0,C 180,E1 25115.959,E2 25115.959} C_VEL
LIN {X 0,Y 222.317,Z 1061.534,A -85,B 0,C 180,E1 25129.603,E2 25129.603} C_VEL
LIN {X 0,Y 220.667,Z 1054.837,A -85,B 0,C 180,E1 25138.643,E2 25138.643} C_VEL
LIN {X 0,Y 249.729,Z 1027.489,A -85,B 0,C 180,E1 25156.776,E2 25156.776} C_VEL
LIN {X 0,Y 291.044,Z 986.912,A -85,B 0,C 180,E1 25169.283,E2 25169.283} C_VEL
LIN {X 0,Y 335.191,Z 933.813,A -85,B 0,C 180,E1 25177.469,E2 25177.469} C_VEL
LIN {X 0,Y 362.006,Z 892.929,A -85,B 0,C 180,E1 25181.31,E2 25181.31} C_VEL
LIN {X 0,Y 362.082,Z 874.219,A -85,B 0,C 180,E1 25189.801,E2 25189.801} C_VEL
LIN {X 0,Y 362.118,Z 866.858,A -85,B 0,C 180,E1 25198.773,E2 25198.773} C_VEL
LIN {X 0,Y 361.835,Z 875.562,A -85,B 0,C 180,E1 25208.416,E2 25208.416} C_VEL
LIN {X 0,Y 361.268,Z 893.106,A -85,B 0,C 180,E1 25216.133,E2 25216.133} C_VEL
LIN {X 0,Y 319.657,Z 952.164,A -85,B 0,C 180,E1 25222.322,E2 25222.322} C_VEL
LIN {X 0,Y 275.143,Z 1000.869,A -85,B 0,C 180,E1 25232.072,E2 25232.072} C_VEL
LIN {X 0,Y 237.265,Z 1036.219,A -85,B 0,C 180,E1 25246.601,E2 25246.601} C_VEL
LIN {X 0,Y 215.634,Z 1057,A -85,B 0,C 180,E1 25265.643,E2 25265.643} C_VEL
LIN {X 0,Y 210.851,Z 1063.316,A -85,B 0,C 180,E1 25283.806,E2 25283.806} C_VEL
LIN {X 0,Y 211.643,Z 1061.578,A -85,B 0,C 180,E1 25296.169,E2 25296.169} C_VEL
LIN {X 0,Y 220.952,Z 1048.402,A -85,B 0,C 180,E1 25315.399,E2 25315.399} C_VEL
LIN {X 0,Y 247.818,Z 1020.266,A -85,B 0,C 180,E1 25332.844,E2 25332.844} C_VEL
LIN {X 0,Y 287.273,Z 977.886,A -85,B 0,C 180,E1 25345.49,E2 25345.49} C_VEL
LIN {X 0,Y 328.65,Z 923.975,A -85,B 0,C 180,E1 25353.747,E2 25353.747} C_VEL
LIN {X 0,Y 352.229,Z 884.663,A -85,B 0,C 180,E1 25357.546,E2 25357.546} C_VEL
LIN {X 0,Y 352.119,Z 861.326,A -85,B 0,C 180,E1 25366.314,E2 25366.314} C_VEL
LIN {X 0,Y 351.371,Z 851.014,A -85,B 0,C 180,E1 25373.827,E2 25373.827} C_VEL
LIN {X 0,Y 352.032,Z 848.054,A -85,B 0,C 180,E1 25378.792,E2 25378.792} C_VEL
LIN {X 0,Y 352.293,Z 858.186,A -85,B 0,C 180,E1 25388.7,E2 25388.7} C_VEL
LIN {X 0,Y 353.627,Z 880.272,A -85,B 0,C 180,E1 25397.868,E2 25397.868} C_VEL
LIN {X 0,Y 352.079,Z 887.53,A -85,B 0,C 180,E1 25399.484,E2 25399.484} C_VEL
LIN {X 0,Y 313.153,Z 947.679,A -85,B 0,C 180,E1 25405.593,E2 25405.593} C_VEL
LIN {X 0,Y 271.581,Z 997.937,A -85,B 0,C 180,E1 25415.255,E2 25415.255} C_VEL
LIN {X 0,Y 235.299,Z 1035.839,A -85,B 0,C 180,E1 25429.876,E2 25429.876} C_VEL
LIN {X 0,Y 215.987,Z 1057.704,A -85,B 0,C 180,E1 25447.286,E2 25447.286} C_VEL
LIN {X 0,Y 211.013,Z 1066.504,A -85,B 0,C 180,E1 25463.813,E2 25463.813} C_VEL
LIN {X 0,Y 211.109,Z 1067.145,A -85,B 0,C 180,E1 25476.186,E2 25476.186} C_VEL
LIN {X 0,Y 216.94,Z 1058.818,A -85,B 0,C 180,E1 25494.071,E2 25494.071} C_VEL
LIN {X 0,Y 220.667,Z 1054.837,A -85,B 0,C 180,E1 25498.643,E2 25498.643} C_VEL
LIN {X 0,Y 222.858,Z 1046.1,A -85,B 0,C 180,E1 25507.529,E2 25507.529} C_VEL
LIN {X 0,Y 258.625,Z 1014.302,A -85,B 0,C 180,E1 25523.371,E2 25523.371} C_VEL
LIN {X 0,Y 303.465,Z 968.956,A -85,B 0,C 180,E1 25534.089,E2 25534.089} C_VEL
LIN {X 0,Y 346.812,Z 913.457,A -85,B 0,C 180,E1 25540.723,E2 25540.723} C_VEL
LIN {X 0,Y 357.06,Z 897.204,A -85,B 0,C 180,E1 25542.185,E2 25542.185} C_VEL
LIN {X 0,Y 357.666,Z 879.924,A -85,B 0,C 180,E1 25550.601,E2 25550.601} C_VEL
LIN {X 0,Y 357.93,Z 873.657,A -85,B 0,C 180,E1 25558.759,E2 25558.759} C_VEL
LIN {X 0,Y 357.308,Z 880.677,A -85,B 0,C 180,E1 25567.295,E2 25567.295} C_VEL
LIN {X 0,Y 356.293,Z 897.136,A -85,B 0,C 180,E1 25575.17,E2 25575.17} C_VEL
LIN {X 0,Y 312.695,Z 956.649,A -85,B 0,C 180,E1 25581.592,E2 25581.592} C_VEL
LIN {X 0,Y 268.306,Z 1003.222,A -85,B 0,C 180,E1 25591.257,E2 25591.257} C_VEL
LIN {X 0,Y 229.566,Z 1037.673,A -85,B 0,C 180,E1 25606.084,E2 25606.084} C_VEL
LIN {X 0,Y 207.251,Z 1057.859,A -85,B 0,C 180,E1 25626.153,E2 25626.153} C_VEL
LIN {X 0,Y 202.85,Z 1063.389,A -85,B 0,C 180,E1 25643.561,E2 25643.561} C_VEL
LIN {X 0,Y 203.686,Z 1061.682,A -85,B 0,C 180,E1 25656.411,E2 25656.411} C_VEL
LIN {X 0,Y 213.609,Z 1048.549,A -85,B 0,C 180,E1 25676.338,E2 25676.338} C_VEL
LIN {X 0,Y 242.223,Z 1020.097,A -85,B 0,C 180,E1 25694.323,E2 25694.323} C_VEL
LIN {X 0,Y 282.596,Z 978.285,A -85,B 0,C 180,E1 25706.824,E2 25706.824} C_VEL
LIN {X 0,Y 325.163,Z 924.304,A -85,B 0,C 180,E1 25715.021,E2 25715.021} C_VEL
LIN {X 0,Y 347.216,Z 889.503,A -85,B 0,C 180,E1 25718.217,E2 25718.217} C_VEL
LIN {X 0,Y 347.702,Z 867.444,A -85,B 0,C 180,E1 25726.779,E2 25726.779} C_VEL
LIN {X 0,Y 347.457,Z 858.098,A -85,B 0,C 180,E1 25733.758,E2 25733.758} C_VEL
LIN {X 0,Y 348.132,Z 855.074,A -85,B 0,C 180,E1 25738.778,E2 25738.778} C_VEL
LIN {X 0,Y 348.138,Z 865.455,A -85,B 0,C 180,E1 25748.804,E2 25748.804} C_VEL
